# B&R Automation Studio project BatteryControl (part 3)

```iecst
	stepTest[0] := 50.000;
	stepTest[1] := 50.000;
	stepTest[2] := 50.000;
	stepTest[3] := 50.000;
	stepTest[4] := 50.000;
	stepTest[5] := 50.000;
	stepTest[6] := 50.000;
	stepTest[7] := 50.000;
	stepTest[8] := 50.000;
	stepTest[9] := 50.000;
	stepTest[10] := 50.010;
	stepTest[11] := 50.010;
	stepTest[12] := 50.010;
	stepTest[13] := 50.010;
	stepTest[14] := 50.010;
	stepTest[15] := 50.010;
	stepTest[16] := 50.010;
	stepTest[17] := 50.010;
	stepTest[18] := 50.010;
	stepTest[19] := 50.010;
	stepTest[20] := 50.010;
	stepTest[21] := 50.010;
	stepTest[22] := 50.010;
	stepTest[23] := 50.010;
	stepTest[24] := 50.010;
	stepTest[25] := 50.010;
	stepTest[26] := 50.010;
	stepTest[27] := 50.010;
	stepTest[28] := 50.010;
	stepTest[29] := 50.010;
	stepTest[30] := 50.010;
	stepTest[31] := 50.010;
	stepTest[32] := 50.010;
	stepTest[33] := 50.010;
	stepTest[34] := 50.010;
	stepTest[35] := 50.010;
	stepTest[36] := 50.010;
	stepTest[37] := 50.010;
	stepTest[38] := 50.010;
	stepTest[39] := 50.010;
	stepTest[40] := 50.000;
	stepTest[41] := 50.000;
	stepTest[42] := 50.000;
	stepTest[43] := 50.000;
	stepTest[44] := 50.000;
	stepTest[45] := 50.000;
	stepTest[46] := 50.000;
	stepTest[47] := 50.000;
	stepTest[48] := 50.000;
	stepTest[49] := 50.000;
	stepTest[50] := 49.990;
	stepTest[51] := 49.990;
	stepTest[52] := 49.990;
	stepTest[53] := 49.990;
	stepTest[54] := 49.990;
	stepTest[55] := 49.990;
	stepTest[56] := 49.990;
	stepTest[57] := 49.990;
	stepTest[58] := 49.990;
	stepTest[59] := 49.990;
	stepTest[60] := 49.990;
	stepTest[61] := 49.990;
	stepTest[62] := 49.990;
	stepTest[63] := 49.990;
	stepTest[64] := 49.990;
	stepTest[65] := 49.990;
	stepTest[66] := 49.990;
	stepTest[67] := 49.990;
	stepTest[68] := 49.990;
	stepTest[69] := 49.990;
	stepTest[70] := 49.990;
	stepTest[71] := 49.990;
	stepTest[72] := 49.990;
	stepTest[73] := 49.990;
	stepTest[74] := 49.990;
	stepTest[75] := 49.990;
	stepTest[76] := 49.990;
	stepTest[77] := 49.990;
	stepTest[78] := 49.990;
	stepTest[79] := 49.990;
	stepTest[80] := 50.000;
	stepTest[81] := 50.000;
	stepTest[82] := 50.000;
	stepTest[83] := 50.000;
	stepTest[84] := 50.000;
	stepTest[85] := 50.000;
	stepTest[86] := 50.000;
	stepTest[87] := 50.000;
	stepTest[88] := 50.000;
	stepTest[89] := 50.000;
	stepTest[90] := 50.020;
	stepTest[91] := 50.020;
	stepTest[92] := 50.020;
	stepTest[93] := 50.020;
	stepTest[94] := 50.020;
	stepTest[95] := 50.020;
	stepTest[96] := 50.020;
	stepTest[97] := 50.020;
	stepTest[98] := 50.020;
	stepTest[99] := 50.020;
	stepTest[100] := 50.020;
	stepTest[101] := 50.020;
	stepTest[102] := 50.020;
	stepTest[103] := 50.020;
	stepTest[104] := 50.020;
	stepTest[105] := 50.020;
	stepTest[106] := 50.020;
	stepTest[107] := 50.020;
	stepTest[108] := 50.020;
	stepTest[109] := 50.020;
	stepTest[110] := 50.020;
	stepTest[111] := 50.020;
	stepTest[112] := 50.020;
	stepTest[113] := 50.020;
	stepTest[114] := 50.020;
	stepTest[115] := 50.020;
	stepTest[116] := 50.020;
	stepTest[117] := 50.020;
	stepTest[118] := 50.020;
	stepTest[119] := 50.020;
	stepTest[120] := 50.000;
	stepTest[121] := 50.000;
	stepTest[122] := 50.000;
	stepTest[123] := 50.000;
	stepTest[124] := 50.000;
	stepTest[125] := 50.000;
	stepTest[126] := 50.000;
	stepTest[127] := 50.000;
	stepTest[128] := 50.000;
	stepTest[129] := 50.000;
	stepTest[130] := 49.980;
	stepTest[131] := 49.980;
	stepTest[132] := 49.980;
	stepTest[133] := 49.980;
	stepTest[134] := 49.980;
	stepTest[135] := 49.980;
	stepTest[136] := 49.980;
	stepTest[137] := 49.980;
	stepTest[138] := 49.980;
	stepTest[139] := 49.980;
	stepTest[140] := 49.980;
	stepTest[141] := 49.980;
	stepTest[142] := 49.980;
	stepTest[143] := 49.980;
	stepTest[144] := 49.980;
	stepTest[145] := 49.980;
	stepTest[146] := 49.980;
	stepTest[147] := 49.980;
	stepTest[148] := 49.980;
	stepTest[149] := 49.980;
	stepTest[150] := 49.980;
	stepTest[151] := 49.980;
	stepTest[152] := 49.980;
	stepTest[153] := 49.980;
	stepTest[154] := 49.980;
	stepTest[155] := 49.980;
	stepTest[156] := 49.980;
	stepTest[157] := 49.980;
	stepTest[158] := 49.980;
	stepTest[159] := 49.980;
	stepTest[160] := 50.000;
	stepTest[161] := 50.000;
	stepTest[162] := 50.000;
	stepTest[163] := 50.000;
	stepTest[164] := 50.000;
	stepTest[165] := 50.000;
	stepTest[166] := 50.000;
	stepTest[167] := 50.000;
	stepTest[168] := 50.000;
	stepTest[169] := 50.000;
	stepTest[170] := 50.100;
	stepTest[171] := 50.100;
	stepTest[172] := 50.100;
	stepTest[173] := 50.100;
	stepTest[174] := 50.100;
	stepTest[175] := 50.100;
	stepTest[176] := 50.100;
	stepTest[177] := 50.100;
	stepTest[178] := 50.100;
	stepTest[179] := 50.100;
	stepTest[180] := 50.100;
	stepTest[181] := 50.100;
	stepTest[182] := 50.100;
	stepTest[183] := 50.100;
	stepTest[184] := 50.100;
	stepTest[185] := 50.100;
	stepTest[186] := 50.100;
	stepTest[187] := 50.100;
	stepTest[188] := 50.100;
	stepTest[189] := 50.100;
	stepTest[190] := 50.100;
	stepTest[191] := 50.100;
	stepTest[192] := 50.100;
	stepTest[193] := 50.100;
	stepTest[194] := 50.100;
	stepTest[195] := 50.100;
	stepTest[196] := 50.100;
	stepTest[197] := 50.100;
	stepTest[198] := 50.100;
	stepTest[199] := 50.100;
	stepTest[200] := 50.000;
	stepTest[201] := 50.000;
	stepTest[202] := 50.000;
	stepTest[203] := 50.000;
	stepTest[204] := 50.000;
	stepTest[205] := 50.000;
	stepTest[206] := 50.000;
	stepTest[207] := 50.000;
	stepTest[208] := 50.000;
	stepTest[209] := 50.000;
	stepTest[210] := 49.900;
	stepTest[211] := 49.900;
	stepTest[212] := 49.900;
	stepTest[213] := 49.900;
	stepTest[214] := 49.900;
	stepTest[215] := 49.900;
	stepTest[216] := 49.900;
	stepTest[217] := 49.900;
	stepTest[218] := 49.900;
	stepTest[219] := 49.900;
	stepTest[220] := 49.900;
	stepTest[221] := 49.900;
	stepTest[222] := 49.900;
	stepTest[223] := 49.900;
	stepTest[224] := 49.900;
	stepTest[225] := 49.900;
	stepTest[226] := 49.900;
	stepTest[227] := 49.900;
	stepTest[228] := 49.900;
	stepTest[229] := 49.900;
	stepTest[230] := 49.900;
	stepTest[231] := 49.900;
	stepTest[232] := 49.900;
	stepTest[233] := 49.900;
	stepTest[234] := 49.900;
	stepTest[235] := 49.900;
	stepTest[236] := 49.900;
	stepTest[237] := 49.900;
	stepTest[238] := 49.900;
	stepTest[239] := 49.900;
	stepTest[240] := 50.000;
	stepTest[241] := 50.000;
	stepTest[242] := 50.000;
	stepTest[243] := 50.000;
	stepTest[244] := 50.000;
	stepTest[245] := 50.000;
	stepTest[246] := 50.000;
	stepTest[247] := 50.000;
	stepTest[248] := 50.000;
	stepTest[249] := 50.000;
	stepTest[250] := 50.200;
	stepTest[251] := 50.200;
	stepTest[252] := 50.200;
	stepTest[253] := 50.200;
	stepTest[254] := 50.200;
	stepTest[255] := 50.200;
	stepTest[256] := 50.200;
	stepTest[257] := 50.200;
	stepTest[258] := 50.200;
	stepTest[259] := 50.200;
	stepTest[260] := 50.200;
	stepTest[261] := 50.200;
	stepTest[262] := 50.200;
	stepTest[263] := 50.200;
	stepTest[264] := 50.200;
	stepTest[265] := 50.200;
	stepTest[266] := 50.200;
	stepTest[267] := 50.200;
	stepTest[268] := 50.200;
	stepTest[269] := 50.200;
	stepTest[270] := 50.200;
	stepTest[271] := 50.200;
	stepTest[272] := 50.200;
	stepTest[273] := 50.200;
	stepTest[274] := 50.200;
	stepTest[275] := 50.200;
	stepTest[276] := 50.200;
	stepTest[277] := 50.200;
	stepTest[278] := 50.200;
	stepTest[279] := 50.200;
	stepTest[280] := 50.000;
	stepTest[281] := 50.000;
	stepTest[282] := 50.000;
	stepTest[283] := 50.000;
	stepTest[284] := 50.000;
	stepTest[285] := 50.000;
	stepTest[286] := 50.000;
	stepTest[287] := 50.000;
	stepTest[288] := 50.000;
	stepTest[289] := 50.000;
	stepTest[290] := 49.800;
	stepTest[291] := 49.800;
	stepTest[292] := 49.800;
	stepTest[293] := 49.800;
	stepTest[294] := 49.800;
	stepTest[295] := 49.800;
	stepTest[296] := 49.800;
	stepTest[297] := 49.800;
	stepTest[298] := 49.800;
	stepTest[299] := 49.800;
	stepTest[300] := 49.800;
	stepTest[301] := 49.800;
	stepTest[302] := 49.800;
	stepTest[303] := 49.800;
	stepTest[304] := 49.800;
	stepTest[305] := 49.800;
	stepTest[306] := 49.800;
	stepTest[307] := 49.800;
	stepTest[308] := 49.800;
	stepTest[309] := 49.800;
	stepTest[310] := 49.800;
	stepTest[311] := 49.800;
	stepTest[312] := 49.800;
	stepTest[313] := 49.800;
	stepTest[314] := 49.800;
	stepTest[315] := 49.800;
	stepTest[316] := 49.800;
	stepTest[317] := 49.800;
	stepTest[318] := 49.800;
	stepTest[319] := 49.800;
	stepTest[320] := 50.000;
	stepTest[321] := 50.000;
	stepTest[322] := 50.000;
	stepTest[323] := 50.000;
	stepTest[324] := 50.000;
	stepTest[325] := 50.000;
	stepTest[326] := 50.000;
	stepTest[327] := 50.000;
	stepTest[328] := 50.000;
	stepTest[329] := 50.000;
	stepTest[330] := 50.300;
	stepTest[331] := 50.300;
	stepTest[332] := 50.300;
	stepTest[333] := 50.300;
	stepTest[334] := 50.300;
	stepTest[335] := 50.300;
	stepTest[336] := 50.300;
	stepTest[337] := 50.300;
	stepTest[338] := 50.300;
	stepTest[339] := 50.300;
	stepTest[340] := 50.300;
	stepTest[341] := 50.300;
	stepTest[342] := 50.300;
	stepTest[343] := 50.300;
	stepTest[344] := 50.300;
	stepTest[345] := 50.300;
	stepTest[346] := 50.300;
	stepTest[347] := 50.300;
	stepTest[348] := 50.300;
	stepTest[349] := 50.300;
	stepTest[350] := 50.300;
	stepTest[351] := 50.300;
	stepTest[352] := 50.300;
	stepTest[353] := 50.300;
	stepTest[354] := 50.300;
	stepTest[355] := 50.300;
	stepTest[356] := 50.300;
	stepTest[357] := 50.300;
	stepTest[358] := 50.300;
	stepTest[359] := 50.300;
	stepTest[360] := 50.000;
	stepTest[361] := 50.000;
	stepTest[362] := 50.000;
	stepTest[363] := 50.000;
	stepTest[364] := 50.000;
	stepTest[365] := 50.000;
	stepTest[366] := 50.000;
	stepTest[367] := 50.000;
	stepTest[368] := 50.000;
	stepTest[369] := 50.000;
	stepTest[370] := 49.700;
	stepTest[371] := 49.700;
	stepTest[372] := 49.700;
	stepTest[373] := 49.700;
	stepTest[374] := 49.700;
	stepTest[375] := 49.700;
	stepTest[376] := 49.700;
	stepTest[377] := 49.700;
	stepTest[378] := 49.700;
	stepTest[379] := 49.700;
	stepTest[380] := 49.700;
	stepTest[381] := 49.700;
	stepTest[382] := 49.700;
	stepTest[383] := 49.700;
	stepTest[384] := 49.700;
	stepTest[385] := 49.700;
	stepTest[386] := 49.700;
	stepTest[387] := 49.700;
	stepTest[388] := 49.700;
	stepTest[389] := 49.700;
	stepTest[390] := 49.700;
	stepTest[391] := 49.700;
	stepTest[392] := 49.700;
	stepTest[393] := 49.700;
	stepTest[394] := 49.700;
	stepTest[395] := 49.700;
	stepTest[396] := 49.700;
	stepTest[397] := 49.700;
	stepTest[398] := 49.700;
	stepTest[399] := 49.700;
	stepTest[400] := 50.000;
	stepTest[401] := 50.000;
	stepTest[402] := 50.000;
	stepTest[403] := 50.000;
	stepTest[404] := 50.000;
	stepTest[405] := 50.000;
	stepTest[406] := 50.000;
	stepTest[407] := 50.000;
	stepTest[408] := 50.000;
	stepTest[409] := 50.000;
	stepTest[410] := 50.400;
	stepTest[411] := 50.400;
	stepTest[412] := 50.400;
	stepTest[413] := 50.400;
	stepTest[414] := 50.400;
	stepTest[415] := 50.400;
	stepTest[416] := 50.400;
	stepTest[417] := 50.400;
	stepTest[418] := 50.400;
	stepTest[419] := 50.400;
	stepTest[420] := 50.400;
	stepTest[421] := 50.400;
	stepTest[422] := 50.400;
	stepTest[423] := 50.400;
	stepTest[424] := 50.400;
	stepTest[425] := 50.400;
	stepTest[426] := 50.400;
	stepTest[427] := 50.400;
	stepTest[428] := 50.400;
	stepTest[429] := 50.400;
	stepTest[430] := 50.400;
	stepTest[431] := 50.400;
	stepTest[432] := 50.400;
	stepTest[433] := 50.400;
	stepTest[434] := 50.400;
	stepTest[435] := 50.400;
	stepTest[436] := 50.400;
	stepTest[437] := 50.400;
	stepTest[438] := 50.400;
	stepTest[439] := 50.400;
	stepTest[440] := 50.000;
	stepTest[441] := 50.000;
	stepTest[442] := 50.000;
	stepTest[443] := 50.000;
	stepTest[444] := 50.000;
	stepTest[445] := 50.000;
	stepTest[446] := 50.000;
	stepTest[447] := 50.000;
	stepTest[448] := 50.000;
	stepTest[449] := 50.000;
	stepTest[450] := 49.600;
	stepTest[451] := 49.600;
	stepTest[452] := 49.600;
	stepTest[453] := 49.600;
	stepTest[454] := 49.600;
	stepTest[455] := 49.600;
	stepTest[456] := 49.600;
	stepTest[457] := 49.600;
	stepTest[458] := 49.600;
	stepTest[459] := 49.600;
	stepTest[460] := 49.600;
	stepTest[461] := 49.600;
	stepTest[462] := 49.600;
	stepTest[463] := 49.600;
	stepTest[464] := 49.600;
	stepTest[465] := 49.600;
	stepTest[466] := 49.600;
	stepTest[467] := 49.600;
	stepTest[468] := 49.600;
	stepTest[469] := 49.600;
	stepTest[470] := 49.600;
	stepTest[471] := 49.600;
	stepTest[472] := 49.600;
	stepTest[473] := 49.600;
	stepTest[474] := 49.600;
	stepTest[475] := 49.600;
	stepTest[476] := 49.600;
	stepTest[477] := 49.600;
	stepTest[478] := 49.600;
	stepTest[479] := 49.600;
	stepTest[480] := 50.000;
	stepTest[481] := 50.000;
	stepTest[482] := 50.000;
	stepTest[483] := 50.000;
	stepTest[484] := 50.000;
	stepTest[485] := 50.000;
	stepTest[486] := 50.000;
	stepTest[487] := 50.000;
	stepTest[488] := 50.000;
	stepTest[489] := 50.000;
	stepTest[490] := 50.500;
	stepTest[491] := 50.500;
	stepTest[492] := 50.500;
	stepTest[493] := 50.500;
	stepTest[494] := 50.500;
	stepTest[495] := 50.500;
	stepTest[496] := 50.500;
	stepTest[497] := 50.500;
	stepTest[498] := 50.500;
	stepTest[499] := 50.500;
	stepTest[500] := 50.500;
	stepTest[501] := 50.500;
	stepTest[502] := 50.500;
	stepTest[503] := 50.500;
	stepTest[504] := 50.500;
	stepTest[505] := 50.500;
	stepTest[506] := 50.500;
	stepTest[507] := 50.500;
	stepTest[508] := 50.500;
	stepTest[509] := 50.500;
	stepTest[510] := 50.500;
	stepTest[511] := 50.500;
	stepTest[512] := 50.500;
	stepTest[513] := 50.500;
	stepTest[514] := 50.500;
	stepTest[515] := 50.500;
	stepTest[516] := 50.500;
	stepTest[517] := 50.500;
	stepTest[518] := 50.500;
	stepTest[519] := 50.500;
	stepTest[520] := 50.000;
	stepTest[521] := 50.000;
	stepTest[522] := 50.000;
	stepTest[523] := 50.000;
	stepTest[524] := 50.000;
	stepTest[525] := 50.000;
	stepTest[526] := 50.000;
	stepTest[527] := 50.000;
	stepTest[528] := 50.000;
	stepTest[529] := 50.000;
	stepTest[530] := 49.500;
	stepTest[531] := 49.500;
	stepTest[532] := 49.500;
	stepTest[533] := 49.500;
	stepTest[534] := 49.500;
	stepTest[535] := 49.500;
	stepTest[536] := 49.500;
	stepTest[537] := 49.500;
	stepTest[538] := 49.500;
	stepTest[539] := 49.500;
	stepTest[540] := 49.500;
	stepTest[541] := 49.500;
	stepTest[542] := 49.500;
	stepTest[543] := 49.500;
	stepTest[544] := 49.500;
	stepTest[545] := 49.500;
	stepTest[546] := 49.500;
	stepTest[547] := 49.500;
	stepTest[548] := 49.500;
	stepTest[549] := 49.500;
	stepTest[550] := 49.500;
	stepTest[551] := 49.500;
	stepTest[552] := 49.500;
	stepTest[553] := 49.500;
	stepTest[554] := 49.500;
	stepTest[555] := 49.500;
	stepTest[556] := 49.500;
	stepTest[557] := 49.500;
	stepTest[558] := 49.500;
	stepTest[559] := 49.500;
	stepTest[560] := 50.000;
	stepTest[561] := 50.000;
	stepTest[562] := 50.000;
	stepTest[563] := 50.000;
	stepTest[564] := 50.000;
	stepTest[565] := 50.000;
	stepTest[566] := 50.000;
	stepTest[567] := 50.000;
	stepTest[568] := 50.000;
	stepTest[569] := 50.000;

	sustainLF[0]:=50.000;
	sustainLF[1]:=50.000;
	sustainLF[2]:=50.000;
	sustainLF[3]:=50.000;
	sustainLF[4]:=50.000;
	sustainLF[5]:=50.000;
	sustainLF[6]:=50.000;
	sustainLF[7]:=50.000;
	sustainLF[8]:=50.000;
	sustainLF[9]:=50.000;
	sustainLF[10]:=50.000;
	sustainLF[11]:=50.000;
	sustainLF[12]:=50.000;
	sustainLF[13]:=50.000;
	sustainLF[14]:=50.000;
	sustainLF[15]:=50.000;
	sustainLF[16]:=50.000;
	sustainLF[17]:=50.000;
	sustainLF[18]:=50.000;
	sustainLF[19]:=50.000;
	sustainLF[20]:=50.000;
	sustainLF[21]:=50.000;
	sustainLF[22]:=50.000;
	sustainLF[23]:=50.000;
	sustainLF[24]:=50.000;
	sustainLF[25]:=50.000;
	sustainLF[26]:=50.000;
	sustainLF[27]:=50.000;
	sustainLF[28]:=50.000;
	sustainLF[29]:=50.000;
	sustainLF[30]:=49.400;
	sustainLF[31]:=49.400;
	sustainLF[32]:=49.400;
	sustainLF[33]:=49.400;
	sustainLF[34]:=49.400;
	sustainLF[35]:=49.400;
	sustainLF[36]:=49.400;
	sustainLF[37]:=49.400;
	sustainLF[38]:=49.400;
	sustainLF[39]:=49.400;
	sustainLF[40]:=49.400;
	sustainLF[41]:=49.400;
	sustainLF[42]:=49.400;
	sustainLF[43]:=49.400;
	sustainLF[44]:=49.400;
	sustainLF[45]:=49.400;
	sustainLF[46]:=49.400;
	sustainLF[47]:=49.400;
	sustainLF[48]:=49.400;
	sustainLF[49]:=49.400;
	sustainLF[50]:=49.400;
	sustainLF[51]:=49.400;
	sustainLF[52]:=49.400;
	sustainLF[53]:=49.400;
	sustainLF[54]:=49.400;
	sustainLF[55]:=49.400;
	sustainLF[56]:=49.400;
	sustainLF[57]:=49.400;
	sustainLF[58]:=49.400;
	sustainLF[59]:=49.400;
	sustainLF[60]:=49.400;
	sustainLF[61]:=49.400;
	sustainLF[62]:=49.400;
	sustainLF[63]:=49.400;
	sustainLF[64]:=49.400;
	sustainLF[65]:=49.400;
	sustainLF[66]:=49.400;
	sustainLF[67]:=49.400;
	sustainLF[68]:=49.400;
	sustainLF[69]:=49.400;
	sustainLF[70]:=49.400;
	sustainLF[71]:=49.400;
	sustainLF[72]:=49.400;
	sustainLF[73]:=49.400;
	sustainLF[74]:=49.400;
	sustainLF[75]:=49.400;
	sustainLF[76]:=49.400;
	sustainLF[77]:=49.400;
	sustainLF[78]:=49.400;
	sustainLF[79]:=49.400;
	sustainLF[80]:=49.400;
	sustainLF[81]:=49.400;
	sustainLF[82]:=49.400;
	sustainLF[83]:=49.400;
	sustainLF[84]:=49.400;
	sustainLF[85]:=49.400;
	sustainLF[86]:=49.400;
	sustainLF[87]:=49.400;
	sustainLF[88]:=49.400;
	sustainLF[89]:=49.400;
	sustainLF[90]:=49.400;
	sustainLF[91]:=49.400;
	sustainLF[92]:=49.400;
	sustainLF[93]:=49.400;
	sustainLF[94]:=49.400;
	sustainLF[95]:=49.400;
	sustainLF[96]:=49.400;
	sustainLF[97]:=49.400;
	sustainLF[98]:=49.400;
	sustainLF[99]:=49.400;
	sustainLF[100]:=49.400;
	sustainLF[101]:=49.400;
	sustainLF[102]:=49.400;
	sustainLF[103]:=49.400;
	sustainLF[104]:=49.400;
	sustainLF[105]:=49.400;
	sustainLF[106]:=49.400;
	sustainLF[107]:=49.400;
	sustainLF[108]:=49.400;
	sustainLF[109]:=49.400;
	sustainLF[110]:=49.400;
	sustainLF[111]:=49.400;
	sustainLF[112]:=49.400;
	sustainLF[113]:=49.400;
	sustainLF[114]:=49.400;
	sustainLF[115]:=49.400;
	sustainLF[116]:=49.400;
	sustainLF[117]:=49.400;
	sustainLF[118]:=49.400;
	sustainLF[119]:=49.400;
	sustainLF[120]:=49.400;
	sustainLF[121]:=49.400;
	sustainLF[122]:=49.400;
	sustainLF[123]:=49.400;
	sustainLF[124]:=49.400;
	sustainLF[125]:=49.400;
	sustainLF[126]:=49.400;
	sustainLF[127]:=49.400;
	sustainLF[128]:=49.400;
	sustainLF[129]:=49.400;
	sustainLF[130]:=49.400;
	sustainLF[131]:=49.400;
	sustainLF[132]:=49.400;
	sustainLF[133]:=49.400;
	sustainLF[134]:=49.400;
	sustainLF[135]:=49.400;
	sustainLF[136]:=49.400;
	sustainLF[137]:=49.400;
	sustainLF[138]:=49.400;
	sustainLF[139]:=49.400;
	sustainLF[140]:=49.400;
	sustainLF[141]:=49.400;
	sustainLF[142]:=49.400;
	sustainLF[143]:=49.400;
	sustainLF[144]:=49.400;
	sustainLF[145]:=49.400;
	sustainLF[146]:=49.400;
	sustainLF[147]:=49.400;
	sustainLF[148]:=49.400;
	sustainLF[149]:=49.400;
	sustainLF[150]:=49.400;
	sustainLF[151]:=49.400;
	sustainLF[152]:=49.400;
	sustainLF[153]:=49.400;
	sustainLF[154]:=49.400;
	sustainLF[155]:=49.400;
	sustainLF[156]:=49.400;
	sustainLF[157]:=49.400;
	sustainLF[158]:=49.400;
	sustainLF[159]:=49.400;
	sustainLF[160]:=49.400;
	sustainLF[161]:=49.400;
	sustainLF[162]:=49.400;
	sustainLF[163]:=49.400;
	sustainLF[164]:=49.400;
	sustainLF[165]:=49.400;
	sustainLF[166]:=49.400;
	sustainLF[167]:=49.400;
	sustainLF[168]:=49.400;
	sustainLF[169]:=49.400;
	sustainLF[170]:=49.400;
	sustainLF[171]:=49.400;
	sustainLF[172]:=49.400;
	sustainLF[173]:=49.400;
	sustainLF[174]:=49.400;
	sustainLF[175]:=49.400;
	sustainLF[176]:=49.400;
	sustainLF[177]:=49.400;
	sustainLF[178]:=49.400;
	sustainLF[179]:=49.400;
	sustainLF[180]:=49.400;
	sustainLF[181]:=49.400;
	sustainLF[182]:=49.400;
	sustainLF[183]:=49.400;
	sustainLF[184]:=49.400;
	sustainLF[185]:=49.400;
	sustainLF[186]:=49.400;
	sustainLF[187]:=49.400;
	sustainLF[188]:=49.400;
	sustainLF[189]:=49.400;
	sustainLF[190]:=49.400;
	sustainLF[191]:=49.400;
	sustainLF[192]:=49.400;
	sustainLF[193]:=49.400;
	sustainLF[194]:=49.400;
	sustainLF[195]:=49.400;
	sustainLF[196]:=49.400;
	sustainLF[197]:=49.400;
	sustainLF[198]:=49.400;
	sustainLF[199]:=49.400;
	sustainLF[200]:=49.400;
	sustainLF[201]:=49.400;
	sustainLF[202]:=49.400;
	sustainLF[203]:=49.400;
	sustainLF[204]:=49.400;
	sustainLF[205]:=49.400;
	sustainLF[206]:=49.400;
	sustainLF[207]:=49.400;
	sustainLF[208]:=49.400;
	sustainLF[209]:=49.400;
	sustainLF[210]:=49.400;
	sustainLF[211]:=49.400;
	sustainLF[212]:=49.400;
	sustainLF[213]:=49.400;
	sustainLF[214]:=49.400;
	sustainLF[215]:=49.400;
	sustainLF[216]:=49.400;
	sustainLF[217]:=49.400;
	sustainLF[218]:=49.400;
	sustainLF[219]:=49.400;
	sustainLF[220]:=49.400;
	sustainLF[221]:=49.400;
	sustainLF[222]:=49.400;
	sustainLF[223]:=49.400;
	sustainLF[224]:=49.400;
	sustainLF[225]:=49.400;
	sustainLF[226]:=49.400;
	sustainLF[227]:=49.400;
	sustainLF[228]:=49.400;
	sustainLF[229]:=49.400;
	sustainLF[230]:=49.400;
	sustainLF[231]:=49.400;
	sustainLF[232]:=49.400;
	sustainLF[233]:=49.400;
	sustainLF[234]:=49.400;
	sustainLF[235]:=49.400;
	sustainLF[236]:=49.400;
	sustainLF[237]:=49.400;
	sustainLF[238]:=49.400;
	sustainLF[239]:=49.400;
	sustainLF[240]:=49.400;
	sustainLF[241]:=49.400;
	sustainLF[242]:=49.400;
	sustainLF[243]:=49.400;
	sustainLF[244]:=49.400;
	sustainLF[245]:=49.400;
	sustainLF[246]:=49.400;
	sustainLF[247]:=49.400;
	sustainLF[248]:=49.400;
	sustainLF[249]:=49.400;
	sustainLF[250]:=49.400;
	sustainLF[251]:=49.400;
	sustainLF[252]:=49.400;
	sustainLF[253]:=49.400;
	sustainLF[254]:=49.400;
	sustainLF[255]:=49.400;
	sustainLF[256]:=49.400;
	sustainLF[257]:=49.400;
	sustainLF[258]:=49.400;
	sustainLF[259]:=49.400;
	sustainLF[260]:=49.400;
	sustainLF[261]:=49.400;
	sustainLF[262]:=49.400;
	sustainLF[263]:=49.400;
	sustainLF[264]:=49.400;
	sustainLF[265]:=49.400;
	sustainLF[266]:=49.400;
	sustainLF[267]:=49.400;
	sustainLF[268]:=49.400;
	sustainLF[269]:=49.400;
	sustainLF[270]:=49.400;
	sustainLF[271]:=49.400;
	sustainLF[272]:=49.400;
	sustainLF[273]:=49.400;
	sustainLF[274]:=49.400;
	sustainLF[275]:=49.400;
	sustainLF[276]:=49.400;
	sustainLF[277]:=49.400;
	sustainLF[278]:=49.400;
	sustainLF[279]:=49.400;
	sustainLF[280]:=49.400;
	sustainLF[281]:=49.400;
	sustainLF[282]:=49.400;
	sustainLF[283]:=49.400;
	sustainLF[284]:=49.400;
	sustainLF[285]:=49.400;
	sustainLF[286]:=49.400;
	sustainLF[287]:=49.400;
	sustainLF[288]:=49.400;
	sustainLF[289]:=49.400;
	sustainLF[290]:=49.400;
	sustainLF[291]:=49.400;
	sustainLF[292]:=49.400;
	sustainLF[293]:=49.400;
	sustainLF[294]:=49.400;
	sustainLF[295]:=49.400;
	sustainLF[296]:=49.400;
	sustainLF[297]:=49.400;
	sustainLF[298]:=49.400;
	sustainLF[299]:=49.400;
	sustainLF[300]:=49.400;
	sustainLF[301]:=49.400;
	sustainLF[302]:=49.400;
	sustainLF[303]:=49.400;
	sustainLF[304]:=49.400;
	sustainLF[305]:=49.400;
	sustainLF[306]:=49.400;
	sustainLF[307]:=49.400;
	sustainLF[308]:=49.400;
	sustainLF[309]:=49.400;
	sustainLF[310]:=49.400;
	sustainLF[311]:=49.400;
	sustainLF[312]:=49.400;
	sustainLF[313]:=49.400;
	sustainLF[314]:=49.400;
	sustainLF[315]:=49.400;
	sustainLF[316]:=49.400;
	sustainLF[317]:=49.400;
	sustainLF[318]:=49.400;
	sustainLF[319]:=49.400;
	sustainLF[320]:=49.400;
	sustainLF[321]:=49.400;
	sustainLF[322]:=49.400;
	sustainLF[323]:=49.400;
	sustainLF[324]:=49.400;
	sustainLF[325]:=49.400;
	sustainLF[326]:=49.400;
	sustainLF[327]:=49.400;
	sustainLF[328]:=49.400;
	sustainLF[329]:=49.400;
	sustainLF[330]:=49.400;
	sustainLF[331]:=49.400;
	sustainLF[332]:=49.400;
	sustainLF[333]:=49.400;
	sustainLF[334]:=49.400;
	sustainLF[335]:=49.400;
	sustainLF[336]:=49.400;
	sustainLF[337]:=49.400;
	sustainLF[338]:=49.400;
	sustainLF[339]:=49.400;
	sustainLF[340]:=49.400;
	sustainLF[341]:=49.400;
	sustainLF[342]:=49.400;
	sustainLF[343]:=49.400;
	sustainLF[344]:=49.400;
	sustainLF[345]:=49.400;
	sustainLF[346]:=49.400;
	sustainLF[347]:=49.400;
	sustainLF[348]:=49.400;
	sustainLF[349]:=49.400;
	sustainLF[350]:=49.400;
	sustainLF[351]:=49.400;
	sustainLF[352]:=49.400;
	sustainLF[353]:=49.400;
	sustainLF[354]:=49.400;
	sustainLF[355]:=49.400;
	sustainLF[356]:=49.400;
	sustainLF[357]:=49.400;
	sustainLF[358]:=49.400;
	sustainLF[359]:=49.400;
	sustainLF[360]:=49.400;
	sustainLF[361]:=49.400;
	sustainLF[362]:=49.400;
	sustainLF[363]:=49.400;
	sustainLF[364]:=49.400;
	sustainLF[365]:=49.400;
	sustainLF[366]:=49.400;
	sustainLF[367]:=49.400;
	sustainLF[368]:=49.400;
	sustainLF[369]:=49.400;
	sustainLF[370]:=49.400;
	sustainLF[371]:=49.400;
	sustainLF[372]:=49.400;
	sustainLF[373]:=49.400;
	sustainLF[374]:=49.400;
	sustainLF[375]:=49.400;
	sustainLF[376]:=49.400;
	sustainLF[377]:=49.400;
	sustainLF[378]:=49.400;
	sustainLF[379]:=49.400;
	sustainLF[380]:=49.400;
	sustainLF[381]:=49.400;
	sustainLF[382]:=49.400;
	sustainLF[383]:=49.400;
	sustainLF[384]:=49.400;
	sustainLF[385]:=49.400;
	sustainLF[386]:=49.400;
	sustainLF[387]:=49.400;
	sustainLF[388]:=49.400;
	sustainLF[389]:=49.400;
	sustainLF[390]:=49.400;
	sustainLF[391]:=49.400;
	sustainLF[392]:=49.400;
	sustainLF[393]:=49.400;
	sustainLF[394]:=49.400;
	sustainLF[395]:=49.400;
	sustainLF[396]:=49.400;
	sustainLF[397]:=49.400;
	sustainLF[398]:=49.400;
	sustainLF[399]:=49.400;
	sustainLF[400]:=49.400;
	sustainLF[401]:=49.400;
	sustainLF[402]:=49.400;
	sustainLF[403]:=49.400;
	sustainLF[404]:=49.400;
	sustainLF[405]:=49.400;
	sustainLF[406]:=49.400;
	sustainLF[407]:=49.400;
	sustainLF[408]:=49.400;
	sustainLF[409]:=49.400;
	sustainLF[410]:=49.400;
	sustainLF[411]:=49.400;
	sustainLF[412]:=49.400;
	sustainLF[413]:=49.400;
	sustainLF[414]:=49.400;
	sustainLF[415]:=49.400;
	sustainLF[416]:=49.400;
	sustainLF[417]:=49.400;
	sustainLF[418]:=49.400;
	sustainLF[419]:=49.400;
	sustainLF[420]:=49.400;
	sustainLF[421]:=49.400;
	sustainLF[422]:=49.400;
	sustainLF[423]:=49.400;
	sustainLF[424]:=49.400;
	sustainLF[425]:=49.400;
	sustainLF[426]:=49.400;
	sustainLF[427]:=49.400;
	sustainLF[428]:=49.400;
	sustainLF[429]:=49.400;
	sustainLF[430]:=49.400;
	sustainLF[431]:=49.400;
	sustainLF[432]:=49.400;
	sustainLF[433]:=49.400;
	sustainLF[434]:=49.400;
	sustainLF[435]:=49.400;
	sustainLF[436]:=49.400;
	sustainLF[437]:=49.400;
	sustainLF[438]:=49.400;
	sustainLF[439]:=49.400;
	sustainLF[440]:=49.400;
	sustainLF[441]:=49.400;
	sustainLF[442]:=49.400;
	sustainLF[443]:=49.400;
	sustainLF[444]:=49.400;
	sustainLF[445]:=49.400;
	sustainLF[446]:=49.400;
	sustainLF[447]:=49.400;
	sustainLF[448]:=49.400;
	sustainLF[449]:=49.400;
	sustainLF[450]:=49.400;
	sustainLF[451]:=49.400;
	sustainLF[452]:=49.400;
	sustainLF[453]:=49.400;
	sustainLF[454]:=49.400;
	sustainLF[455]:=49.400;
	sustainLF[456]:=49.400;
	sustainLF[457]:=49.400;
	sustainLF[458]:=49.400;
	sustainLF[459]:=49.400;
	sustainLF[460]:=49.400;
	sustainLF[461]:=49.400;
	sustainLF[462]:=49.400;
	sustainLF[463]:=49.400;
	sustainLF[464]:=49.400;
	sustainLF[465]:=49.400;
	sustainLF[466]:=49.400;
	sustainLF[467]:=49.400;
	sustainLF[468]:=49.400;
	sustainLF[469]:=49.400;
	sustainLF[470]:=49.400;
	sustainLF[471]:=49.400;
	sustainLF[472]:=49.400;
	sustainLF[473]:=49.400;
	sustainLF[474]:=49.400;
	sustainLF[475]:=49.400;
	sustainLF[476]:=49.400;
	sustainLF[477]:=49.400;
	sustainLF[478]:=49.400;
	sustainLF[479]:=49.400;
	sustainLF[480]:=49.400;
	sustainLF[481]:=49.400;
	sustainLF[482]:=49.400;
	sustainLF[483]:=49.400;
	sustainLF[484]:=49.400;
	sustainLF[485]:=49.400;
	sustainLF[486]:=49.400;
	sustainLF[487]:=49.400;
	sustainLF[488]:=49.400;
	sustainLF[489]:=49.400;
	sustainLF[490]:=49.400;
	sustainLF[491]:=49.400;
	sustainLF[492]:=49.400;
	sustainLF[493]:=49.400;
	sustainLF[494]:=49.400;
	sustainLF[495]:=49.400;
	sustainLF[496]:=49.400;
	sustainLF[497]:=49.400;
	sustainLF[498]:=49.400;
	sustainLF[499]:=49.400;
	sustainLF[500]:=49.400;
	sustainLF[501]:=49.400;
	sustainLF[502]:=49.400;
	sustainLF[503]:=49.400;
	sustainLF[504]:=49.400;
	sustainLF[505]:=49.400;
	sustainLF[506]:=49.400;
	sustainLF[507]:=49.400;
	sustainLF[508]:=49.400;
	sustainLF[509]:=49.400;
	sustainLF[510]:=49.400;
	sustainLF[511]:=49.400;
	sustainLF[512]:=49.400;
	sustainLF[513]:=49.400;
	sustainLF[514]:=49.400;
	sustainLF[515]:=49.400;
	sustainLF[516]:=49.400;
	sustainLF[517]:=49.400;
	sustainLF[518]:=49.400;
	sustainLF[519]:=49.400;
	sustainLF[520]:=49.400;
	sustainLF[521]:=49.400;
	sustainLF[522]:=49.400;
	sustainLF[523]:=49.400;
	sustainLF[524]:=49.400;
	sustainLF[525]:=49.400;
	sustainLF[526]:=49.400;
	sustainLF[527]:=49.400;
	sustainLF[528]:=49.400;
	sustainLF[529]:=49.400;
	sustainLF[530]:=49.400;
	sustainLF[531]:=49.400;
	sustainLF[532]:=49.400;
	sustainLF[533]:=49.400;
	sustainLF[534]:=49.400;
	sustainLF[535]:=49.400;
	sustainLF[536]:=49.400;
	sustainLF[537]:=49.400;
	sustainLF[538]:=49.400;
	sustainLF[539]:=49.400;
	sustainLF[540]:=49.400;
	sustainLF[541]:=49.400;
	sustainLF[542]:=49.400;
	sustainLF[543]:=49.400;
	sustainLF[544]:=49.400;
	sustainLF[545]:=49.400;
	sustainLF[546]:=49.400;
	sustainLF[547]:=49.400;
	sustainLF[548]:=49.400;
	sustainLF[549]:=49.400;
	sustainLF[550]:=49.400;
	sustainLF[551]:=49.400;
	sustainLF[552]:=49.400;
	sustainLF[553]:=49.400;
	sustainLF[554]:=49.400;
	sustainLF[555]:=49.400;
	sustainLF[556]:=49.400;
	sustainLF[557]:=49.400;
	sustainLF[558]:=49.400;
	sustainLF[559]:=49.400;
	sustainLF[560]:=49.400;
	sustainLF[561]:=49.400;
	sustainLF[562]:=49.400;
	sustainLF[563]:=49.400;
	sustainLF[564]:=49.400;
	sustainLF[565]:=49.400;
	sustainLF[566]:=49.400;
	sustainLF[567]:=49.400;
	sustainLF[568]:=49.400;
	sustainLF[569]:=49.400;
	sustainLF[570]:=49.400;
	sustainLF[571]:=49.400;
	sustainLF[572]:=49.400;
	sustainLF[573]:=49.400;
	sustainLF[574]:=49.400;
	sustainLF[575]:=49.400;
	sustainLF[576]:=49.400;
	sustainLF[577]:=49.400;
	sustainLF[578]:=49.400;
	sustainLF[579]:=49.400;
	sustainLF[580]:=49.400;
	sustainLF[581]:=49.400;
	sustainLF[582]:=49.400;
	sustainLF[583]:=49.400;
	sustainLF[584]:=49.400;
	sustainLF[585]:=49.400;
	sustainLF[586]:=49.400;
	sustainLF[587]:=49.400;
	sustainLF[588]:=49.400;
	sustainLF[589]:=49.400;
	sustainLF[590]:=49.400;
	sustainLF[591]:=49.400;
	sustainLF[592]:=49.400;
	sustainLF[593]:=49.400;
	sustainLF[594]:=49.400;
	sustainLF[595]:=49.400;
	sustainLF[596]:=49.400;
	sustainLF[597]:=49.400;
	sustainLF[598]:=49.400;
	sustainLF[599]:=49.400;
	sustainLF[600]:=49.400;
	sustainLF[601]:=49.400;
	sustainLF[602]:=49.400;
	sustainLF[603]:=49.400;
	sustainLF[604]:=49.400;
	sustainLF[605]:=49.400;
	sustainLF[606]:=49.400;
	sustainLF[607]:=49.400;
	sustainLF[608]:=49.400;
	sustainLF[609]:=49.400;
	sustainLF[610]:=49.400;
	sustainLF[611]:=49.400;
	sustainLF[612]:=49.400;
	sustainLF[613]:=49.400;
	sustainLF[614]:=49.400;
	sustainLF[615]:=49.400;
	sustainLF[616]:=49.400;
	sustainLF[617]:=49.400;
	sustainLF[618]:=49.400;
	sustainLF[619]:=49.400;
	sustainLF[620]:=49.400;
	sustainLF[621]:=49.400;
	sustainLF[622]:=49.400;
	sustainLF[623]:=49.400;
	sustainLF[624]:=49.400;
	sustainLF[625]:=49.400;
	sustainLF[626]:=49.400;
	sustainLF[627]:=49.400;
	sustainLF[628]:=49.400;
	sustainLF[629]:=49.400;
	sustainLF[630]:=49.400;
	sustainLF[631]:=49.400;
	sustainLF[632]:=49.400;
	sustainLF[633]:=49.400;
	sustainLF[634]:=49.400;
	sustainLF[635]:=49.400;
	sustainLF[636]:=49.400;
	sustainLF[637]:=49.400;
	sustainLF[638]:=49.400;
	sustainLF[639]:=49.400;
	sustainLF[640]:=49.400;
	sustainLF[641]:=49.400;
	sustainLF[642]:=49.400;
	sustainLF[643]:=49.400;
	sustainLF[644]:=49.400;
	sustainLF[645]:=49.400;
	sustainLF[646]:=49.400;
	sustainLF[647]:=49.400;
	sustainLF[648]:=49.400;
	sustainLF[649]:=49.400;
	sustainLF[650]:=49.400;
	sustainLF[651]:=49.400;
	sustainLF[652]:=49.400;
	sustainLF[653]:=49.400;
	sustainLF[654]:=49.400;
	sustainLF[655]:=49.400;
	sustainLF[656]:=49.400;
	sustainLF[657]:=49.400;
	sustainLF[658]:=49.400;
	sustainLF[659]:=49.400;
	sustainLF[660]:=49.400;
	sustainLF[661]:=49.400;
	sustainLF[662]:=49.400;
	sustainLF[663]:=49.400;
	sustainLF[664]:=49.400;
	sustainLF[665]:=49.400;
	sustainLF[666]:=49.400;
	sustainLF[667]:=49.400;
	sustainLF[668]:=49.400;
	sustainLF[669]:=49.400;
	sustainLF[670]:=49.400;
	sustainLF[671]:=49.400;
	sustainLF[672]:=49.400;
	sustainLF[673]:=49.400;
	sustainLF[674]:=49.400;
	sustainLF[675]:=49.400;
	sustainLF[676]:=49.400;
	sustainLF[677]:=49.400;
	sustainLF[678]:=49.400;
	sustainLF[679]:=49.400;
	sustainLF[680]:=49.400;
	sustainLF[681]:=49.400;
	sustainLF[682]:=49.400;
	sustainLF[683]:=49.400;
	sustainLF[684]:=49.400;
	sustainLF[685]:=49.400;
	sustainLF[686]:=49.400;
	sustainLF[687]:=49.400;
	sustainLF[688]:=49.400;
	sustainLF[689]:=49.400;
	sustainLF[690]:=49.400;
	sustainLF[691]:=49.400;
	sustainLF[692]:=49.400;
	sustainLF[693]:=49.400;
	sustainLF[694]:=49.400;
	sustainLF[695]:=49.400;
	sustainLF[696]:=49.400;
	sustainLF[697]:=49.400;
	sustainLF[698]:=49.400;
	sustainLF[699]:=49.400;
	sustainLF[700]:=49.400;
	sustainLF[701]:=49.400;
	sustainLF[702]:=49.400;
	sustainLF[703]:=49.400;
	sustainLF[704]:=49.400;
	sustainLF[705]:=49.400;
	sustainLF[706]:=49.400;
	sustainLF[707]:=49.400;
	sustainLF[708]:=49.400;
	sustainLF[709]:=49.400;
	sustainLF[710]:=49.400;
	sustainLF[711]:=49.400;
	sustainLF[712]:=49.400;
	sustainLF[713]:=49.400;
	sustainLF[714]:=49.400;
	sustainLF[715]:=49.400;
	sustainLF[716]:=49.400;
	sustainLF[717]:=49.400;
	sustainLF[718]:=49.400;
	sustainLF[719]:=49.400;
	sustainLF[720]:=49.400;
	sustainLF[721]:=49.400;
	sustainLF[722]:=49.400;
	sustainLF[723]:=49.400;
	sustainLF[724]:=49.400;
	sustainLF[725]:=49.400;
	sustainLF[726]:=49.400;
	sustainLF[727]:=49.400;
	sustainLF[728]:=49.400;
	sustainLF[729]:=49.400;
	sustainLF[730]:=49.400;
	sustainLF[731]:=49.400;
	sustainLF[732]:=49.400;
	sustainLF[733]:=49.400;
	sustainLF[734]:=49.400;
	sustainLF[735]:=49.400;
	sustainLF[736]:=49.400;
	sustainLF[737]:=49.400;
	sustainLF[738]:=49.400;
	sustainLF[739]:=49.400;
	sustainLF[740]:=49.400;
	sustainLF[741]:=49.400;
	sustainLF[742]:=49.400;
	sustainLF[743]:=49.400;
	sustainLF[744]:=49.400;
	sustainLF[745]:=49.400;
	sustainLF[746]:=49.400;
	sustainLF[747]:=49.400;
	sustainLF[748]:=49.400;
	sustainLF[749]:=49.400;
	sustainLF[750]:=49.400;
	sustainLF[751]:=49.400;
	sustainLF[752]:=49.400;
	sustainLF[753]:=49.400;
	sustainLF[754]:=49.400;
	sustainLF[755]:=49.400;
	sustainLF[756]:=49.400;
	sustainLF[757]:=49.400;
	sustainLF[758]:=49.400;
	sustainLF[759]:=49.400;
	sustainLF[760]:=49.400;
	sustainLF[761]:=49.400;
	sustainLF[762]:=49.400;
	sustainLF[763]:=49.400;
	sustainLF[764]:=49.400;
	sustainLF[765]:=49.400;
	sustainLF[766]:=49.400;
	sustainLF[767]:=49.400;
	sustainLF[768]:=49.400;
	sustainLF[769]:=49.400;
	sustainLF[770]:=49.400;
	sustainLF[771]:=49.400;
	sustainLF[772]:=49.400;
	sustainLF[773]:=49.400;
	sustainLF[774]:=49.400;
	sustainLF[775]:=49.400;
	sustainLF[776]:=49.400;
	sustainLF[777]:=49.400;
	sustainLF[778]:=49.400;
	sustainLF[779]:=49.400;
	sustainLF[780]:=49.400;
	sustainLF[781]:=49.400;
	sustainLF[782]:=49.400;
	sustainLF[783]:=49.400;
	sustainLF[784]:=49.400;
	sustainLF[785]:=49.400;
	sustainLF[786]:=49.400;
	sustainLF[787]:=49.400;
	sustainLF[788]:=49.400;
	sustainLF[789]:=49.400;
	sustainLF[790]:=49.400;
	sustainLF[791]:=49.400;
	sustainLF[792]:=49.400;
	sustainLF[793]:=49.400;
	sustainLF[794]:=49.400;
	sustainLF[795]:=49.400;
	sustainLF[796]:=49.400;
	sustainLF[797]:=49.400;
	sustainLF[798]:=49.400;
	sustainLF[799]:=49.400;
	sustainLF[800]:=49.400;
	sustainLF[801]:=49.400;
	sustainLF[802]:=49.400;
	sustainLF[803]:=49.400;
	sustainLF[804]:=49.400;
	sustainLF[805]:=49.400;
	sustainLF[806]:=49.400;
	sustainLF[807]:=49.400;
	sustainLF[808]:=49.400;
	sustainLF[809]:=49.400;
	sustainLF[810]:=49.400;
	sustainLF[811]:=49.400;
	sustainLF[812]:=49.400;
	sustainLF[813]:=49.400;
	sustainLF[814]:=49.400;
	sustainLF[815]:=49.400;
	sustainLF[816]:=49.400;
	sustainLF[817]:=49.400;
	sustainLF[818]:=49.400;
	sustainLF[819]:=49.400;
	sustainLF[820]:=49.400;
	sustainLF[821]:=49.400;
	sustainLF[822]:=49.400;
	sustainLF[823]:=49.400;
	sustainLF[824]:=49.400;
	sustainLF[825]:=49.400;
	sustainLF[826]:=49.400;
	sustainLF[827]:=49.400;
	sustainLF[828]:=49.400;
	sustainLF[829]:=49.400;
	sustainLF[830]:=49.400;
	sustainLF[831]:=49.400;
	sustainLF[832]:=49.400;
	sustainLF[833]:=49.400;
	sustainLF[834]:=49.400;
	sustainLF[835]:=49.400;
	sustainLF[836]:=49.400;
	sustainLF[837]:=49.400;
	sustainLF[838]:=49.400;
	sustainLF[839]:=49.400;
	sustainLF[840]:=49.400;
	sustainLF[841]:=49.400;
	sustainLF[842]:=49.400;
	sustainLF[843]:=49.400;
	sustainLF[844]:=49.400;
	sustainLF[845]:=49.400;
	sustainLF[846]:=49.400;
	sustainLF[847]:=49.400;
	sustainLF[848]:=49.400;
	sustainLF[849]:=49.400;
	sustainLF[850]:=49.400;
	sustainLF[851]:=49.400;
	sustainLF[852]:=49.400;
	sustainLF[853]:=49.400;
	sustainLF[854]:=49.400;
	sustainLF[855]:=49.400;
	sustainLF[856]:=49.400;
	sustainLF[857]:=49.400;
	sustainLF[858]:=49.400;
	sustainLF[859]:=49.400;
	sustainLF[860]:=49.400;
	sustainLF[861]:=49.400;
	sustainLF[862]:=49.400;
	sustainLF[863]:=49.400;
	sustainLF[864]:=49.400;
	sustainLF[865]:=49.400;
	sustainLF[866]:=49.400;
	sustainLF[867]:=49.400;
	sustainLF[868]:=49.400;
	sustainLF[869]:=49.400;
	sustainLF[870]:=49.400;
	sustainLF[871]:=49.400;
	sustainLF[872]:=49.400;
	sustainLF[873]:=49.400;
	sustainLF[874]:=49.400;
	sustainLF[875]:=49.400;
	sustainLF[876]:=49.400;
	sustainLF[877]:=49.400;
	sustainLF[878]:=49.400;
	sustainLF[879]:=49.400;
	sustainLF[880]:=49.400;
	sustainLF[881]:=49.400;
	sustainLF[882]:=49.400;
	sustainLF[883]:=49.400;
	sustainLF[884]:=49.400;
	sustainLF[885]:=49.400;
	sustainLF[886]:=49.400;
	sustainLF[887]:=49.400;
	sustainLF[888]:=49.400;
	sustainLF[889]:=49.400;
	sustainLF[890]:=49.400;
	sustainLF[891]:=49.400;
	sustainLF[892]:=49.400;
	sustainLF[893]:=49.400;
	sustainLF[894]:=49.400;
	sustainLF[895]:=49.400;
	sustainLF[896]:=49.400;
	sustainLF[897]:=49.400;
	sustainLF[898]:=49.400;
	sustainLF[899]:=49.400;
	sustainLF[900]:=49.400;
	sustainLF[901]:=49.400;
	sustainLF[902]:=49.400;
	sustainLF[903]:=49.400;
	sustainLF[904]:=49.400;
	sustainLF[905]:=49.400;
	sustainLF[906]:=49.400;
	sustainLF[907]:=49.400;
	sustainLF[908]:=49.400;
	sustainLF[909]:=49.400;
	sustainLF[910]:=49.400;
	sustainLF[911]:=49.400;
	sustainLF[912]:=49.400;
	sustainLF[913]:=49.400;
	sustainLF[914]:=49.400;
	sustainLF[915]:=49.400;
	sustainLF[916]:=49.400;
	sustainLF[917]:=49.400;
	sustainLF[918]:=49.400;
	sustainLF[919]:=49.400;
	sustainLF[920]:=49.400;
	sustainLF[921]:=49.400;
	sustainLF[922]:=49.400;
	sustainLF[923]:=49.400;
	sustainLF[924]:=49.400;
	sustainLF[925]:=49.400;
	sustainLF[926]:=49.400;
	sustainLF[927]:=49.400;
	sustainLF[928]:=49.400;
	sustainLF[929]:=49.400;
	sustainLF[930]:=50.000;
	sustainLF[931]:=50.000;
	sustainLF[932]:=50.000;
	sustainLF[933]:=50.000;
	sustainLF[934]:=50.000;
	sustainLF[935]:=50.000;
	sustainLF[936]:=50.000;
	sustainLF[937]:=50.000;
	sustainLF[938]:=50.000;
	sustainLF[939]:=50.000;
	sustainLF[940]:=50.000;
	sustainLF[941]:=50.000;
	sustainLF[942]:=50.000;
	sustainLF[943]:=50.000;
	sustainLF[944]:=50.000;
	sustainLF[945]:=50.000;
	sustainLF[946]:=50.000;
	sustainLF[947]:=50.000;
	sustainLF[948]:=50.000;
	sustainLF[949]:=50.000;
	sustainLF[950]:=50.000;
	sustainLF[951]:=50.000;
	sustainLF[952]:=50.000;
	sustainLF[953]:=50.000;
	sustainLF[954]:=50.000;
	sustainLF[955]:=50.000;
	sustainLF[956]:=50.000;
	sustainLF[957]:=50.000;
	sustainLF[958]:=50.000;
	sustainLF[959]:=50.000;

	stepTestFull[0]:=50.000;
	stepTestFull[1]:=50.000;
	stepTestFull[2]:=50.000;
	stepTestFull[3]:=50.000;
	stepTestFull[4]:=50.000;
	stepTestFull[5]:=50.000;
	stepTestFull[6]:=50.000;
	stepTestFull[7]:=50.000;
	stepTestFull[8]:=50.000;
	stepTestFull[9]:=50.000;
	stepTestFull[10]:=50.000;
	stepTestFull[11]:=50.000;
	stepTestFull[12]:=50.000;
	stepTestFull[13]:=50.000;
	stepTestFull[14]:=50.000;
	stepTestFull[15]:=50.000;
	stepTestFull[16]:=50.000;
	stepTestFull[17]:=50.000;
	stepTestFull[18]:=50.000;
	stepTestFull[19]:=50.000;
	stepTestFull[20]:=50.000;
	stepTestFull[21]:=50.000;
	stepTestFull[22]:=50.000;
	stepTestFull[23]:=50.000;
	stepTestFull[24]:=50.000;
	stepTestFull[25]:=50.000;
	stepTestFull[26]:=50.000;
	stepTestFull[27]:=50.000;
	stepTestFull[28]:=50.000;
	stepTestFull[29]:=50.000;
	stepTestFull[30]:=50.010;
	stepTestFull[31]:=50.010;
	stepTestFull[32]:=50.010;
	stepTestFull[33]:=50.010;
	stepTestFull[34]:=50.010;
	stepTestFull[35]:=50.010;
	stepTestFull[36]:=50.010;
	stepTestFull[37]:=50.010;
	stepTestFull[38]:=50.010;
	stepTestFull[39]:=50.010;
	stepTestFull[40]:=50.010;
	stepTestFull[41]:=50.010;
	stepTestFull[42]:=50.010;
	stepTestFull[43]:=50.010;
	stepTestFull[44]:=50.010;
	stepTestFull[45]:=50.010;
	stepTestFull[46]:=50.010;
	stepTestFull[47]:=50.010;
	stepTestFull[48]:=50.010;
	stepTestFull[49]:=50.010;
	stepTestFull[50]:=50.010;
	stepTestFull[51]:=50.010;
	stepTestFull[52]:=50.010;
	stepTestFull[53]:=50.010;
	stepTestFull[54]:=50.010;
	stepTestFull[55]:=50.010;
	stepTestFull[56]:=50.010;
	stepTestFull[57]:=50.010;
	stepTestFull[58]:=50.010;
	stepTestFull[59]:=50.010;
	stepTestFull[60]:=50.010;
	stepTestFull[61]:=50.010;
	stepTestFull[62]:=50.010;
	stepTestFull[63]:=50.010;
	stepTestFull[64]:=50.010;
	stepTestFull[65]:=50.010;
	stepTestFull[66]:=50.010;
	stepTestFull[67]:=50.010;
	stepTestFull[68]:=50.010;
	stepTestFull[69]:=50.010;
	stepTestFull[70]:=50.010;
	stepTestFull[71]:=50.010;
	stepTestFull[72]:=50.010;
	stepTestFull[73]:=50.010;
	stepTestFull[74]:=50.010;
	stepTestFull[75]:=50.010;
	stepTestFull[76]:=50.010;
	stepTestFull[77]:=50.010;
	stepTestFull[78]:=50.010;
	stepTestFull[79]:=50.010;
	stepTestFull[80]:=50.010;
	stepTestFull[81]:=50.010;
	stepTestFull[82]:=50.010;
	stepTestFull[83]:=50.010;
	stepTestFull[84]:=50.010;
	stepTestFull[85]:=50.010;
	stepTestFull[86]:=50.010;
	stepTestFull[87]:=50.010;
	stepTestFull[88]:=50.010;
	stepTestFull[89]:=50.010;
	stepTestFull[90]:=50.010;
	stepTestFull[91]:=50.010;
	stepTestFull[92]:=50.010;
	stepTestFull[93]:=50.010;
	stepTestFull[94]:=50.010;
	stepTestFull[95]:=50.010;
	stepTestFull[96]:=50.010;
	stepTestFull[97]:=50.010;
	stepTestFull[98]:=50.010;
	stepTestFull[99]:=50.010;
	stepTestFull[100]:=50.010;
	stepTestFull[101]:=50.010;
	stepTestFull[102]:=50.010;
	stepTestFull[103]:=50.010;
	stepTestFull[104]:=50.010;
	stepTestFull[105]:=50.010;
	stepTestFull[106]:=50.010;
	stepTestFull[107]:=50.010;
	stepTestFull[108]:=50.010;
	stepTestFull[109]:=50.010;
	stepTestFull[110]:=50.010;
	stepTestFull[111]:=50.010;
	stepTestFull[112]:=50.010;
	stepTestFull[113]:=50.010;
	stepTestFull[114]:=50.010;
	stepTestFull[115]:=50.010;
	stepTestFull[116]:=50.010;
	stepTestFull[117]:=50.010;
	stepTestFull[118]:=50.010;
	stepTestFull[119]:=50.010;
	stepTestFull[120]:=50.010;
	stepTestFull[121]:=50.010;
	stepTestFull[122]:=50.010;
	stepTestFull[123]:=50.010;
	stepTestFull[124]:=50.010;
	stepTestFull[125]:=50.010;
	stepTestFull[126]:=50.010;
	stepTestFull[127]:=50.010;
	stepTestFull[128]:=50.010;
	stepTestFull[129]:=50.010;
	stepTestFull[130]:=50.010;
	stepTestFull[131]:=50.010;
	stepTestFull[132]:=50.010;
	stepTestFull[133]:=50.010;
	stepTestFull[134]:=50.010;
	stepTestFull[135]:=50.010;
	stepTestFull[136]:=50.010;
	stepTestFull[137]:=50.010;
	stepTestFull[138]:=50.010;
	stepTestFull[139]:=50.010;
	stepTestFull[140]:=50.010;
	stepTestFull[141]:=50.010;
	stepTestFull[142]:=50.010;
	stepTestFull[143]:=50.010;
	stepTestFull[144]:=50.010;
	stepTestFull[145]:=50.010;
	stepTestFull[146]:=50.010;
	stepTestFull[147]:=50.010;
	stepTestFull[148]:=50.010;
	stepTestFull[149]:=50.010;
	stepTestFull[150]:=50.010;
	stepTestFull[151]:=50.010;
	stepTestFull[152]:=50.010;
	stepTestFull[153]:=50.010;
	stepTestFull[154]:=50.010;
	stepTestFull[155]:=50.010;
	stepTestFull[156]:=50.010;
	stepTestFull[157]:=50.010;
	stepTestFull[158]:=50.010;
	stepTestFull[159]:=50.010;
	stepTestFull[160]:=50.010;
	stepTestFull[161]:=50.010;
	stepTestFull[162]:=50.010;
	stepTestFull[163]:=50.010;
	stepTestFull[164]:=50.010;
	stepTestFull[165]:=50.010;
	stepTestFull[166]:=50.010;
	stepTestFull[167]:=50.010;
	stepTestFull[168]:=50.010;
	stepTestFull[169]:=50.010;
	stepTestFull[170]:=50.010;
	stepTestFull[171]:=50.010;
	stepTestFull[172]:=50.010;
	stepTestFull[173]:=50.010;
	stepTestFull[174]:=50.010;
	stepTestFull[175]:=50.010;
	stepTestFull[176]:=50.010;
	stepTestFull[177]:=50.010;
	stepTestFull[178]:=50.010;
	stepTestFull[179]:=50.010;
	stepTestFull[180]:=50.010;
	stepTestFull[181]:=50.010;
	stepTestFull[182]:=50.010;
	stepTestFull[183]:=50.010;
	stepTestFull[184]:=50.010;
	stepTestFull[185]:=50.010;
	stepTestFull[186]:=50.010;
	stepTestFull[187]:=50.010;
	stepTestFull[188]:=50.010;
	stepTestFull[189]:=50.010;
	stepTestFull[190]:=50.010;
	stepTestFull[191]:=50.010;
	stepTestFull[192]:=50.010;
	stepTestFull[193]:=50.010;
	stepTestFull[194]:=50.010;
	stepTestFull[195]:=50.010;
	stepTestFull[196]:=50.010;
	stepTestFull[197]:=50.010;
	stepTestFull[198]:=50.010;
	stepTestFull[199]:=50.010;
	stepTestFull[200]:=50.010;
	stepTestFull[201]:=50.010;
	stepTestFull[202]:=50.010;
	stepTestFull[203]:=50.010;
	stepTestFull[204]:=50.010;
	stepTestFull[205]:=50.010;
	stepTestFull[206]:=50.010;
	stepTestFull[207]:=50.010;
	stepTestFull[208]:=50.010;
	stepTestFull[209]:=50.010;
	stepTestFull[210]:=50.000;
	stepTestFull[211]:=50.000;
	stepTestFull[212]:=50.000;
	stepTestFull[213]:=50.000;
	stepTestFull[214]:=50.000;
	stepTestFull[215]:=50.000;
	stepTestFull[216]:=50.000;
	stepTestFull[217]:=50.000;
	stepTestFull[218]:=50.000;
	stepTestFull[219]:=50.000;
	stepTestFull[220]:=50.000;
	stepTestFull[221]:=50.000;
	stepTestFull[222]:=50.000;
	stepTestFull[223]:=50.000;
	stepTestFull[224]:=50.000;
	stepTestFull[225]:=50.000;
	stepTestFull[226]:=50.000;
	stepTestFull[227]:=50.000;
	stepTestFull[228]:=50.000;
	stepTestFull[229]:=50.000;
	stepTestFull[230]:=50.000;
	stepTestFull[231]:=50.000;
	stepTestFull[232]:=50.000;
	stepTestFull[233]:=50.000;
	stepTestFull[234]:=50.000;
	stepTestFull[235]:=50.000;
	stepTestFull[236]:=50.000;
	stepTestFull[237]:=50.000;
	stepTestFull[238]:=50.000;
	stepTestFull[239]:=50.000;
	stepTestFull[240]:=50.000;
	stepTestFull[241]:=50.000;
	stepTestFull[242]:=50.000;
	stepTestFull[243]:=50.000;
	stepTestFull[244]:=50.000;
	stepTestFull[245]:=50.000;
	stepTestFull[246]:=50.000;
	stepTestFull[247]:=50.000;
	stepTestFull[248]:=50.000;
	stepTestFull[249]:=50.000;
	stepTestFull[250]:=50.000;
	stepTestFull[251]:=50.000;
	stepTestFull[252]:=50.000;
	stepTestFull[253]:=50.000;
	stepTestFull[254]:=50.000;
	stepTestFull[255]:=50.000;
	stepTestFull[256]:=50.000;
	stepTestFull[257]:=50.000;
	stepTestFull[258]:=50.000;
	stepTestFull[259]:=50.000;
	stepTestFull[260]:=50.000;
	stepTestFull[261]:=50.000;
	stepTestFull[262]:=50.000;
	stepTestFull[263]:=50.000;
	stepTestFull[264]:=50.000;
	stepTestFull[265]:=50.000;
	stepTestFull[266]:=50.000;
	stepTestFull[267]:=50.000;
	stepTestFull[268]:=50.000;
	stepTestFull[269]:=50.000;
	stepTestFull[270]:=49.990;
	stepTestFull[271]:=49.990;
	stepTestFull[272]:=49.990;
	stepTestFull[273]:=49.990;
	stepTestFull[274]:=49.990;
	stepTestFull[275]:=49.990;
	stepTestFull[276]:=49.990;
	stepTestFull[277]:=49.990;
	stepTestFull[278]:=49.990;
	stepTestFull[279]:=49.990;
	stepTestFull[280]:=49.990;
	stepTestFull[281]:=49.990;
	stepTestFull[282]:=49.990;
	stepTestFull[283]:=49.990;
	stepTestFull[284]:=49.990;
	stepTestFull[285]:=49.990;
	stepTestFull[286]:=49.990;
	stepTestFull[287]:=49.990;
	stepTestFull[288]:=49.990;
	stepTestFull[289]:=49.990;
	stepTestFull[290]:=49.990;
	stepTestFull[291]:=49.990;
	stepTestFull[292]:=49.990;
	stepTestFull[293]:=49.990;
	stepTestFull[294]:=49.990;
	stepTestFull[295]:=49.990;
	stepTestFull[296]:=49.990;
	stepTestFull[297]:=49.990;
	stepTestFull[298]:=49.990;
	stepTestFull[299]:=49.990;
	stepTestFull[300]:=49.990;
	stepTestFull[301]:=49.990;
	stepTestFull[302]:=49.990;
	stepTestFull[303]:=49.990;
	stepTestFull[304]:=49.990;
	stepTestFull[305]:=49.990;
	stepTestFull[306]:=49.990;
	stepTestFull[307]:=49.990;
	stepTestFull[308]:=49.990;
	stepTestFull[309]:=49.990;
	stepTestFull[310]:=49.990;
	stepTestFull[311]:=49.990;
	stepTestFull[312]:=49.990;
	stepTestFull[313]:=49.990;
	stepTestFull[314]:=49.990;
	stepTestFull[315]:=49.990;
	stepTestFull[316]:=49.990;
	stepTestFull[317]:=49.990;
	stepTestFull[318]:=49.990;
	stepTestFull[319]:=49.990;
	stepTestFull[320]:=49.990;
	stepTestFull[321]:=49.990;
	stepTestFull[322]:=49.990;
	stepTestFull[323]:=49.990;
	stepTestFull[324]:=49.990;
	stepTestFull[325]:=49.990;
	stepTestFull[326]:=49.990;
	stepTestFull[327]:=49.990;
	stepTestFull[328]:=49.990;
	stepTestFull[329]:=49.990;
	stepTestFull[330]:=49.990;
	stepTestFull[331]:=49.990;
	stepTestFull[332]:=49.990;
	stepTestFull[333]:=49.990;
	stepTestFull[334]:=49.990;
	stepTestFull[335]:=49.990;
	stepTestFull[336]:=49.990;
	stepTestFull[337]:=49.990;
	stepTestFull[338]:=49.990;
	stepTestFull[339]:=49.990;
	stepTestFull[340]:=49.990;
	stepTestFull[341]:=49.990;
	stepTestFull[342]:=49.990;
	stepTestFull[343]:=49.990;
	stepTestFull[344]:=49.990;
	stepTestFull[345]:=49.990;
	stepTestFull[346]:=49.990;
	stepTestFull[347]:=49.990;
	stepTestFull[348]:=49.990;
	stepTestFull[349]:=49.990;
	stepTestFull[350]:=49.990;
	stepTestFull[351]:=49.990;
	stepTestFull[352]:=49.990;
	stepTestFull[353]:=49.990;
	stepTestFull[354]:=49.990;
	stepTestFull[355]:=49.990;
	stepTestFull[356]:=49.990;
	stepTestFull[357]:=49.990;
	stepTestFull[358]:=49.990;
	stepTestFull[359]:=49.990;
	stepTestFull[360]:=49.990;
	stepTestFull[361]:=49.990;
	stepTestFull[362]:=49.990;
	stepTestFull[363]:=49.990;
	stepTestFull[364]:=49.990;
	stepTestFull[365]:=49.990;
	stepTestFull[366]:=49.990;
	stepTestFull[367]:=49.990;
	stepTestFull[368]:=49.990;
	stepTestFull[369]:=49.990;
	stepTestFull[370]:=49.990;
	stepTestFull[371]:=49.990;
	stepTestFull[372]:=49.990;
	stepTestFull[373]:=49.990;
	stepTestFull[374]:=49.990;
	stepTestFull[375]:=49.990;
	stepTestFull[376]:=49.990;
	stepTestFull[377]:=49.990;
	stepTestFull[378]:=49.990;
	stepTestFull[379]:=49.990;
	stepTestFull[380]:=49.990;
	stepTestFull[381]:=49.990;
	stepTestFull[382]:=49.990;
	stepTestFull[383]:=49.990;
	stepTestFull[384]:=49.990;
	stepTestFull[385]:=49.990;
	stepTestFull[386]:=49.990;
	stepTestFull[387]:=49.990;
	stepTestFull[388]:=49.990;
	stepTestFull[389]:=49.990;
	stepTestFull[390]:=49.990;
	stepTestFull[391]:=49.990;
	stepTestFull[392]:=49.990;
	stepTestFull[393]:=49.990;
	stepTestFull[394]:=49.990;
	stepTestFull[395]:=49.990;
	stepTestFull[396]:=49.990;
	stepTestFull[397]:=49.990;
	stepTestFull[398]:=49.990;
	stepTestFull[399]:=49.990;
	stepTestFull[400]:=49.990;
	stepTestFull[401]:=49.990;
	stepTestFull[402]:=49.990;
	stepTestFull[403]:=49.990;
	stepTestFull[404]:=49.990;
	stepTestFull[405]:=49.990;
	stepTestFull[406]:=49.990;
	stepTestFull[407]:=49.990;
	stepTestFull[408]:=49.990;
	stepTestFull[409]:=49.990;
	stepTestFull[410]:=49.990;
	stepTestFull[411]:=49.990;
	stepTestFull[412]:=49.990;
	stepTestFull[413]:=49.990;
	stepTestFull[414]:=49.990;
	stepTestFull[415]:=49.990;
	stepTestFull[416]:=49.990;
	stepTestFull[417]:=49.990;
	stepTestFull[418]:=49.990;
	stepTestFull[419]:=49.990;
	stepTestFull[420]:=49.990;
	stepTestFull[421]:=49.990;
	stepTestFull[422]:=49.990;
	stepTestFull[423]:=49.990;
	stepTestFull[424]:=49.990;
	stepTestFull[425]:=49.990;
	stepTestFull[426]:=49.990;
	stepTestFull[427]:=49.990;
	stepTestFull[428]:=49.990;
	stepTestFull[429]:=49.990;
	stepTestFull[430]:=49.990;
	stepTestFull[431]:=49.990;
	stepTestFull[432]:=49.990;
	stepTestFull[433]:=49.990;
	stepTestFull[434]:=49.990;
	stepTestFull[435]:=49.990;
	stepTestFull[436]:=49.990;
	stepTestFull[437]:=49.990;
	stepTestFull[438]:=49.990;
	stepTestFull[439]:=49.990;
	stepTestFull[440]:=49.990;
	stepTestFull[441]:=49.990;
	stepTestFull[442]:=49.990;
	stepTestFull[443]:=49.990;
	stepTestFull[444]:=49.990;
	stepTestFull[445]:=49.990;
	stepTestFull[446]:=49.990;
	stepTestFull[447]:=49.990;
	stepTestFull[448]:=49.990;
	stepTestFull[449]:=49.990;
	stepTestFull[450]:=50.000;
	stepTestFull[451]:=50.000;
	stepTestFull[452]:=50.000;
	stepTestFull[453]:=50.000;
	stepTestFull[454]:=50.000;
	stepTestFull[455]:=50.000;
	stepTestFull[456]:=50.000;
	stepTestFull[457]:=50.000;
	stepTestFull[458]:=50.000;
	stepTestFull[459]:=50.000;
	stepTestFull[460]:=50.000;
	stepTestFull[461]:=50.000;
	stepTestFull[462]:=50.000;
	stepTestFull[463]:=50.000;
	stepTestFull[464]:=50.000;
	stepTestFull[465]:=50.000;
	stepTestFull[466]:=50.000;
	stepTestFull[467]:=50.000;
	stepTestFull[468]:=50.000;
	stepTestFull[469]:=50.000;
	stepTestFull[470]:=50.000;
	stepTestFull[471]:=50.000;
	stepTestFull[472]:=50.000;
	stepTestFull[473]:=50.000;
	stepTestFull[474]:=50.000;
	stepTestFull[475]:=50.000;
	stepTestFull[476]:=50.000;
	stepTestFull[477]:=50.000;
	stepTestFull[478]:=50.000;
	stepTestFull[479]:=50.000;
	stepTestFull[480]:=50.000;
	stepTestFull[481]:=50.000;
	stepTestFull[482]:=50.000;
	stepTestFull[483]:=50.000;
	stepTestFull[484]:=50.000;
	stepTestFull[485]:=50.000;
	stepTestFull[486]:=50.000;
	stepTestFull[487]:=50.000;
	stepTestFull[488]:=50.000;
	stepTestFull[489]:=50.000;
	stepTestFull[490]:=50.000;
	stepTestFull[491]:=50.000;
	stepTestFull[492]:=50.000;
	stepTestFull[493]:=50.000;
	stepTestFull[494]:=50.000;
	stepTestFull[495]:=50.000;
	stepTestFull[496]:=50.000;
	stepTestFull[497]:=50.000;
	stepTestFull[498]:=50.000;
	stepTestFull[499]:=50.000;
	stepTestFull[500]:=50.000;
	stepTestFull[501]:=50.000;
	stepTestFull[502]:=50.000;
	stepTestFull[503]:=50.000;
	stepTestFull[504]:=50.000;
	stepTestFull[505]:=50.000;
	stepTestFull[506]:=50.000;
	stepTestFull[507]:=50.000;
	stepTestFull[508]:=50.000;
	stepTestFull[509]:=50.000;
	stepTestFull[510]:=50.020;
	stepTestFull[511]:=50.020;
	stepTestFull[512]:=50.020;
	stepTestFull[513]:=50.020;
	stepTestFull[514]:=50.020;
	stepTestFull[515]:=50.020;
	stepTestFull[516]:=50.020;
	stepTestFull[517]:=50.020;
	stepTestFull[518]:=50.020;
	stepTestFull[519]:=50.020;
	stepTestFull[520]:=50.020;
	stepTestFull[521]:=50.020;
	stepTestFull[522]:=50.020;
	stepTestFull[523]:=50.020;
	stepTestFull[524]:=50.020;
	stepTestFull[525]:=50.020;
	stepTestFull[526]:=50.020;
	stepTestFull[527]:=50.020;
	stepTestFull[528]:=50.020;
	stepTestFull[529]:=50.020;
	stepTestFull[530]:=50.020;
	stepTestFull[531]:=50.020;
	stepTestFull[532]:=50.020;
	stepTestFull[533]:=50.020;
	stepTestFull[534]:=50.020;
	stepTestFull[535]:=50.020;
	stepTestFull[536]:=50.020;
	stepTestFull[537]:=50.020;
	stepTestFull[538]:=50.020;
	stepTestFull[539]:=50.020;
	stepTestFull[540]:=50.020;
	stepTestFull[541]:=50.020;
	stepTestFull[542]:=50.020;
	stepTestFull[543]:=50.020;
	stepTestFull[544]:=50.020;
	stepTestFull[545]:=50.020;
	stepTestFull[546]:=50.020;
	stepTestFull[547]:=50.020;
	stepTestFull[548]:=50.020;
	stepTestFull[549]:=50.020;
	stepTestFull[550]:=50.020;
	stepTestFull[551]:=50.020;
	stepTestFull[552]:=50.020;
	stepTestFull[553]:=50.020;
	stepTestFull[554]:=50.020;
	stepTestFull[555]:=50.020;
	stepTestFull[556]:=50.020;
	stepTestFull[557]:=50.020;
	stepTestFull[558]:=50.020;
	stepTestFull[559]:=50.020;
	stepTestFull[560]:=50.020;
	stepTestFull[561]:=50.020;
	stepTestFull[562]:=50.020;
	stepTestFull[563]:=50.020;
	stepTestFull[564]:=50.020;
	stepTestFull[565]:=50.020;
	stepTestFull[566]:=50.020;
	stepTestFull[567]:=50.020;
	stepTestFull[568]:=50.020;
	stepTestFull[569]:=50.020;
	stepTestFull[570]:=50.020;
	stepTestFull[571]:=50.020;
	stepTestFull[572]:=50.020;
	stepTestFull[573]:=50.020;
	stepTestFull[574]:=50.020;
	stepTestFull[575]:=50.020;
	stepTestFull[576]:=50.020;
	stepTestFull[577]:=50.020;
	stepTestFull[578]:=50.020;
	stepTestFull[579]:=50.020;
	stepTestFull[580]:=50.020;
	stepTestFull[581]:=50.020;
	stepTestFull[582]:=50.020;
	stepTestFull[583]:=50.020;
	stepTestFull[584]:=50.020;
	stepTestFull[585]:=50.020;
	stepTestFull[586]:=50.020;
	stepTestFull[587]:=50.020;
	stepTestFull[588]:=50.020;
	stepTestFull[589]:=50.020;
	stepTestFull[590]:=50.020;
	stepTestFull[591]:=50.020;
	stepTestFull[592]:=50.020;
	stepTestFull[593]:=50.020;
	stepTestFull[594]:=50.020;
	stepTestFull[595]:=50.020;
	stepTestFull[596]:=50.020;
	stepTestFull[597]:=50.020;
	stepTestFull[598]:=50.020;
	stepTestFull[599]:=50.020;
	stepTestFull[600]:=50.020;
	stepTestFull[601]:=50.020;
	stepTestFull[602]:=50.020;
	stepTestFull[603]:=50.020;
	stepTestFull[604]:=50.020;
	stepTestFull[605]:=50.020;
	stepTestFull[606]:=50.020;
	stepTestFull[607]:=50.020;
	stepTestFull[608]:=50.020;
	stepTestFull[609]:=50.020;
	stepTestFull[610]:=50.020;
	stepTestFull[611]:=50.020;
	stepTestFull[612]:=50.020;
	stepTestFull[613]:=50.020;
	stepTestFull[614]:=50.020;
	stepTestFull[615]:=50.020;
	stepTestFull[616]:=50.020;
	stepTestFull[617]:=50.020;
	stepTestFull[618]:=50.020;
	stepTestFull[619]:=50.020;
	stepTestFull[620]:=50.020;
	stepTestFull[621]:=50.020;
	stepTestFull[622]:=50.020;
	stepTestFull[623]:=50.020;
	stepTestFull[624]:=50.020;
	stepTestFull[625]:=50.020;
	stepTestFull[626]:=50.020;
	stepTestFull[627]:=50.020;
	stepTestFull[628]:=50.020;
	stepTestFull[629]:=50.020;
	stepTestFull[630]:=50.020;
	stepTestFull[631]:=50.020;
	stepTestFull[632]:=50.020;
	stepTestFull[633]:=50.020;
	stepTestFull[634]:=50.020;
	stepTestFull[635]:=50.020;
	stepTestFull[636]:=50.020;
	stepTestFull[637]:=50.020;
	stepTestFull[638]:=50.020;
	stepTestFull[639]:=50.020;
	stepTestFull[640]:=50.020;
	stepTestFull[641]:=50.020;
	stepTestFull[642]:=50.020;
	stepTestFull[643]:=50.020;
	stepTestFull[644]:=50.020;
	stepTestFull[645]:=50.020;
	stepTestFull[646]:=50.020;
	stepTestFull[647]:=50.020;
	stepTestFull[648]:=50.020;
	stepTestFull[649]:=50.020;
	stepTestFull[650]:=50.020;
	stepTestFull[651]:=50.020;
	stepTestFull[652]:=50.020;
	stepTestFull[653]:=50.020;
	stepTestFull[654]:=50.020;
	stepTestFull[655]:=50.020;
	stepTestFull[656]:=50.020;
	stepTestFull[657]:=50.020;
	stepTestFull[658]:=50.020;
	stepTestFull[659]:=50.020;
	stepTestFull[660]:=50.020;
	stepTestFull[661]:=50.020;
	stepTestFull[662]:=50.020;
	stepTestFull[663]:=50.020;
	stepTestFull[664]:=50.020;
	stepTestFull[665]:=50.020;
	stepTestFull[666]:=50.020;
	stepTestFull[667]:=50.020;
	stepTestFull[668]:=50.020;
	stepTestFull[669]:=50.020;
	stepTestFull[670]:=50.020;
	stepTestFull[671]:=50.020;
	stepTestFull[672]:=50.020;
	stepTestFull[673]:=50.020;
	stepTestFull[674]:=50.020;
	stepTestFull[675]:=50.020;
	stepTestFull[676]:=50.020;
	stepTestFull[677]:=50.020;
	stepTestFull[678]:=50.020;
	stepTestFull[679]:=50.020;
	stepTestFull[680]:=50.020;
	stepTestFull[681]:=50.020;
	stepTestFull[682]:=50.020;
	stepTestFull[683]:=50.020;
	stepTestFull[684]:=50.020;
	stepTestFull[685]:=50.020;
	stepTestFull[686]:=50.020;
	stepTestFull[687]:=50.020;
	stepTestFull[688]:=50.020;
	stepTestFull[689]:=50.020;
	stepTestFull[690]:=50.000;
	stepTestFull[691]:=50.000;
	stepTestFull[692]:=50.000;
	stepTestFull[693]:=50.000;
	stepTestFull[694]:=50.000;
	stepTestFull[695]:=50.000;
	stepTestFull[696]:=50.000;
	stepTestFull[697]:=50.000;
	stepTestFull[698]:=50.000;
	stepTestFull[699]:=50.000;
	stepTestFull[700]:=50.000;
	stepTestFull[701]:=50.000;
	stepTestFull[702]:=50.000;
	stepTestFull[703]:=50.000;
	stepTestFull[704]:=50.000;
	stepTestFull[705]:=50.000;
	stepTestFull[706]:=50.000;
	stepTestFull[707]:=50.000;
	stepTestFull[708]:=50.000;
	stepTestFull[709]:=50.000;
	stepTestFull[710]:=50.000;
	stepTestFull[711]:=50.000;
	stepTestFull[712]:=50.000;
	stepTestFull[713]:=50.000;
	stepTestFull[714]:=50.000;
	stepTestFull[715]:=50.000;
	stepTestFull[716]:=50.000;
	stepTestFull[717]:=50.000;
	stepTestFull[718]:=50.000;
	stepTestFull[719]:=50.000;
	stepTestFull[720]:=50.000;
	stepTestFull[721]:=50.000;
	stepTestFull[722]:=50.000;
	stepTestFull[723]:=50.000;
	stepTestFull[724]:=50.000;
	stepTestFull[725]:=50.000;
	stepTestFull[726]:=50.000;
	stepTestFull[727]:=50.000;
	stepTestFull[728]:=50.000;
	stepTestFull[729]:=50.000;
	stepTestFull[730]:=50.000;
	stepTestFull[731]:=50.000;
	stepTestFull[732]:=50.000;
	stepTestFull[733]:=50.000;
	stepTestFull[734]:=50.000;
	stepTestFull[735]:=50.000;
	stepTestFull[736]:=50.000;
	stepTestFull[737]:=50.000;
	stepTestFull[738]:=50.000;
	stepTestFull[739]:=50.000;
	stepTestFull[740]:=50.000;
	stepTestFull[741]:=50.000;
	stepTestFull[742]:=50.000;
	stepTestFull[743]:=50.000;
	stepTestFull[744]:=50.000;
	stepTestFull[745]:=50.000;
	stepTestFull[746]:=50.000;
	stepTestFull[747]:=50.000;
	stepTestFull[748]:=50.000;
	stepTestFull[749]:=50.000;
	stepTestFull[750]:=49.980;
	stepTestFull[751]:=49.980;
	stepTestFull[752]:=49.980;
	stepTestFull[753]:=49.980;
	stepTestFull[754]:=49.980;
	stepTestFull[755]:=49.980;
	stepTestFull[756]:=49.980;
	stepTestFull[757]:=49.980;
	stepTestFull[758]:=49.980;
	stepTestFull[759]:=49.980;
	stepTestFull[760]:=49.980;
	stepTestFull[761]:=49.980;
	stepTestFull[762]:=49.980;
	stepTestFull[763]:=49.980;
	stepTestFull[764]:=49.980;
	stepTestFull[765]:=49.980;
	stepTestFull[766]:=49.980;
	stepTestFull[767]:=49.980;
	stepTestFull[768]:=49.980;
	stepTestFull[769]:=49.980;
	stepTestFull[770]:=49.980;
	stepTestFull[771]:=49.980;
	stepTestFull[772]:=49.980;
	stepTestFull[773]:=49.980;
	stepTestFull[774]:=49.980;
	stepTestFull[775]:=49.980;
	stepTestFull[776]:=49.980;
	stepTestFull[777]:=49.980;
	stepTestFull[778]:=49.980;
	stepTestFull[779]:=49.980;
	stepTestFull[780]:=49.980;
	stepTestFull[781]:=49.980;
	stepTestFull[782]:=49.980;
	stepTestFull[783]:=49.980;
	stepTestFull[784]:=49.980;
	stepTestFull[785]:=49.980;
	stepTestFull[786]:=49.980;
	stepTestFull[787]:=49.980;
	stepTestFull[788]:=49.980;
	stepTestFull[789]:=49.980;
	stepTestFull[790]:=49.980;
	stepTestFull[791]:=49.980;
	stepTestFull[792]:=49.980;
	stepTestFull[793]:=49.980;
	stepTestFull[794]:=49.980;
	stepTestFull[795]:=49.980;
	stepTestFull[796]:=49.980;
	stepTestFull[797]:=49.980;
	stepTestFull[798]:=49.980;
	stepTestFull[799]:=49.980;
	stepTestFull[800]:=49.980;
	stepTestFull[801]:=49.980;
	stepTestFull[802]:=49.980;
	stepTestFull[803]:=49.980;
	stepTestFull[804]:=49.980;
	stepTestFull[805]:=49.980;
	stepTestFull[806]:=49.980;
	stepTestFull[807]:=49.980;
	stepTestFull[808]:=49.980;
	stepTestFull[809]:=49.980;
	stepTestFull[810]:=49.980;
	stepTestFull[811]:=49.980;
	stepTestFull[812]:=49.980;
	stepTestFull[813]:=49.980;
	stepTestFull[814]:=49.980;
	stepTestFull[815]:=49.980;
	stepTestFull[816]:=49.980;
	stepTestFull[817]:=49.980;
	stepTestFull[818]:=49.980;
	stepTestFull[819]:=49.980;
	stepTestFull[820]:=49.980;
	stepTestFull[821]:=49.980;
	stepTestFull[822]:=49.980;
	stepTestFull[823]:=49.980;
	stepTestFull[824]:=49.980;
	stepTestFull[825]:=49.980;
	stepTestFull[826]:=49.980;
	stepTestFull[827]:=49.980;
	stepTestFull[828]:=49.980;
	stepTestFull[829]:=49.980;
	stepTestFull[830]:=49.980;
	stepTestFull[831]:=49.980;
	stepTestFull[832]:=49.980;
	stepTestFull[833]:=49.980;
	stepTestFull[834]:=49.980;
	stepTestFull[835]:=49.980;
	stepTestFull[836]:=49.980;
	stepTestFull[837]:=49.980;
	stepTestFull[838]:=49.980;
	stepTestFull[839]:=49.980;
	stepTestFull[840]:=49.980;
	stepTestFull[841]:=49.980;
	stepTestFull[842]:=49.980;
	stepTestFull[843]:=49.980;
	stepTestFull[844]:=49.980;
	stepTestFull[845]:=49.980;
	stepTestFull[846]:=49.980;
	stepTestFull[847]:=49.980;
	stepTestFull[848]:=49.980;
	stepTestFull[849]:=49.980;
	stepTestFull[850]:=49.980;
	stepTestFull[851]:=49.980;
	stepTestFull[852]:=49.980;
	stepTestFull[853]:=49.980;
	stepTestFull[854]:=49.980;
	stepTestFull[855]:=49.980;
	stepTestFull[856]:=49.980;
	stepTestFull[857]:=49.980;
	stepTestFull[858]:=49.980;
	stepTestFull[859]:=49.980;
	stepTestFull[860]:=49.980;
	stepTestFull[861]:=49.980;
	stepTestFull[862]:=49.980;
	stepTestFull[863]:=49.980;
	stepTestFull[864]:=49.980;
	stepTestFull[865]:=49.980;
	stepTestFull[866]:=49.980;
	stepTestFull[867]:=49.980;
	stepTestFull[868]:=49.980;
	stepTestFull[869]:=49.980;
	stepTestFull[870]:=49.980;
	stepTestFull[871]:=49.980;
	stepTestFull[872]:=49.980;
	stepTestFull[873]:=49.980;
	stepTestFull[874]:=49.980;
	stepTestFull[875]:=49.980;
	stepTestFull[876]:=49.980;
	stepTestFull[877]:=49.980;
	stepTestFull[878]:=49.980;
	stepTestFull[879]:=49.980;
	stepTestFull[880]:=49.980;
	stepTestFull[881]:=49.980;
	stepTestFull[882]:=49.980;
	stepTestFull[883]:=49.980;
	stepTestFull[884]:=49.980;
	stepTestFull[885]:=49.980;
	stepTestFull[886]:=49.980;
	stepTestFull[887]:=49.980;
	stepTestFull[888]:=49.980;
	stepTestFull[889]:=49.980;
	stepTestFull[890]:=49.980;
	stepTestFull[891]:=49.980;
	stepTestFull[892]:=49.980;
	stepTestFull[893]:=49.980;
	stepTestFull[894]:=49.980;
	stepTestFull[895]:=49.980;
	stepTestFull[896]:=49.980;
	stepTestFull[897]:=49.980;
	stepTestFull[898]:=49.980;
	stepTestFull[899]:=49.980;
	stepTestFull[900]:=49.980;
	stepTestFull[901]:=49.980;
	stepTestFull[902]:=49.980;
	stepTestFull[903]:=49.980;
	stepTestFull[904]:=49.980;
	stepTestFull[905]:=49.980;
	stepTestFull[906]:=49.980;
	stepTestFull[907]:=49.980;
	stepTestFull[908]:=49.980;
	stepTestFull[909]:=49.980;
	stepTestFull[910]:=49.980;
	stepTestFull[911]:=49.980;
	stepTestFull[912]:=49.980;
	stepTestFull[913]:=49.980;
	stepTestFull[914]:=49.980;
	stepTestFull[915]:=49.980;
	stepTestFull[916]:=49.980;
	stepTestFull[917]:=49.980;
	stepTestFull[918]:=49.980;
	stepTestFull[919]:=49.980;
	stepTestFull[920]:=49.980;
	stepTestFull[921]:=49.980;
	stepTestFull[922]:=49.980;
	stepTestFull[923]:=49.980;
	stepTestFull[924]:=49.980;
	stepTestFull[925]:=49.980;
	stepTestFull[926]:=49.980;
	stepTestFull[927]:=49.980;
	stepTestFull[928]:=49.980;
	stepTestFull[929]:=49.980;
	stepTestFull[930]:=50.000;
	stepTestFull[931]:=50.000;
	stepTestFull[932]:=50.000;
	stepTestFull[933]:=50.000;
	stepTestFull[934]:=50.000;
	stepTestFull[935]:=50.000;
	stepTestFull[936]:=50.000;
	stepTestFull[937]:=50.000;
	stepTestFull[938]:=50.000;
	stepTestFull[939]:=50.000;
	stepTestFull[940]:=50.000;
	stepTestFull[941]:=50.000;
	stepTestFull[942]:=50.000;
	stepTestFull[943]:=50.000;
	stepTestFull[944]:=50.000;
	stepTestFull[945]:=50.000;
	stepTestFull[946]:=50.000;
	stepTestFull[947]:=50.000;
	stepTestFull[948]:=50.000;
	stepTestFull[949]:=50.000;
	stepTestFull[950]:=50.000;
	stepTestFull[951]:=50.000;
	stepTestFull[952]:=50.000;
	stepTestFull[953]:=50.000;
	stepTestFull[954]:=50.000;
	stepTestFull[955]:=50.000;
	stepTestFull[956]:=50.000;
	stepTestFull[957]:=50.000;
	stepTestFull[958]:=50.000;
	stepTestFull[959]:=50.000;
	stepTestFull[960]:=50.000;
	stepTestFull[961]:=50.000;
	stepTestFull[962]:=50.000;
	stepTestFull[963]:=50.000;
	stepTestFull[964]:=50.000;
	stepTestFull[965]:=50.000;
	stepTestFull[966]:=50.000;
	stepTestFull[967]:=50.000;
	stepTestFull[968]:=50.000;
	stepTestFull[969]:=50.000;
	stepTestFull[970]:=50.000;
	stepTestFull[971]:=50.000;
	stepTestFull[972]:=50.000;
	stepTestFull[973]:=50.000;
	stepTestFull[974]:=50.000;
	stepTestFull[975]:=50.000;
	stepTestFull[976]:=50.000;
	stepTestFull[977]:=50.000;
	stepTestFull[978]:=50.000;
	stepTestFull[979]:=50.000;
	stepTestFull[980]:=50.000;
	stepTestFull[981]:=50.000;
	stepTestFull[982]:=50.000;
	stepTestFull[983]:=50.000;
	stepTestFull[984]:=50.000;
	stepTestFull[985]:=50.000;
	stepTestFull[986]:=50.000;
	stepTestFull[987]:=50.000;
	stepTestFull[988]:=50.000;
	stepTestFull[989]:=50.000;
	stepTestFull[990]:=50.100;
	stepTestFull[991]:=50.100;
	stepTestFull[992]:=50.100;
	stepTestFull[993]:=50.100;
	stepTestFull[994]:=50.100;
	stepTestFull[995]:=50.100;
	stepTestFull[996]:=50.100;
	stepTestFull[997]:=50.100;
	stepTestFull[998]:=50.100;
	stepTestFull[999]:=50.100;
	stepTestFull[1000]:=50.100;
	stepTestFull[1001]:=50.100;
	stepTestFull[1002]:=50.100;
	stepTestFull[1003]:=50.100;
	stepTestFull[1004]:=50.100;
	stepTestFull[1005]:=50.100;
	stepTestFull[1006]:=50.100;
	stepTestFull[1007]:=50.100;
	stepTestFull[1008]:=50.100;
	stepTestFull[1009]:=50.100;
	stepTestFull[1010]:=50.100;
	stepTestFull[1011]:=50.100;
	stepTestFull[1012]:=50.100;
	stepTestFull[1013]:=50.100;
	stepTestFull[1014]:=50.100;
	stepTestFull[1015]:=50.100;
	stepTestFull[1016]:=50.100;
	stepTestFull[1017]:=50.100;
	stepTestFull[1018]:=50.100;
	stepTestFull[1019]:=50.100;
	stepTestFull[1020]:=50.100;
	stepTestFull[1021]:=50.100;
	stepTestFull[1022]:=50.100;
	stepTestFull[1023]:=50.100;
	stepTestFull[1024]:=50.100;
	stepTestFull[1025]:=50.100;
	stepTestFull[1026]:=50.100;
	stepTestFull[1027]:=50.100;
	stepTestFull[1028]:=50.100;
	stepTestFull[1029]:=50.100;
	stepTestFull[1030]:=50.100;
	stepTestFull[1031]:=50.100;
	stepTestFull[1032]:=50.100;
	stepTestFull[1033]:=50.100;
	stepTestFull[1034]:=50.100;
	stepTestFull[1035]:=50.100;
	stepTestFull[1036]:=50.100;
	stepTestFull[1037]:=50.100;
	stepTestFull[1038]:=50.100;
	stepTestFull[1039]:=50.100;
	stepTestFull[1040]:=50.100;
	stepTestFull[1041]:=50.100;
	stepTestFull[1042]:=50.100;
	stepTestFull[1043]:=50.100;
	stepTestFull[1044]:=50.100;
	stepTestFull[1045]:=50.100;
	stepTestFull[1046]:=50.100;
	stepTestFull[1047]:=50.100;
	stepTestFull[1048]:=50.100;
	stepTestFull[1049]:=50.100;
	stepTestFull[1050]:=50.100;
	stepTestFull[1051]:=50.100;
	stepTestFull[1052]:=50.100;
	stepTestFull[1053]:=50.100;
	stepTestFull[1054]:=50.100;
	stepTestFull[1055]:=50.100;
	stepTestFull[1056]:=50.100;
	stepTestFull[1057]:=50.100;
	stepTestFull[1058]:=50.100;
	stepTestFull[1059]:=50.100;
	stepTestFull[1060]:=50.100;
	stepTestFull[1061]:=50.100;
	stepTestFull[1062]:=50.100;
	stepTestFull[1063]:=50.100;
	stepTestFull[1064]:=50.100;
	stepTestFull[1065]:=50.100;
	stepTestFull[1066]:=50.100;
	stepTestFull[1067]:=50.100;
	stepTestFull[1068]:=50.100;
	stepTestFull[1069]:=50.100;
	stepTestFull[1070]:=50.100;
	stepTestFull[1071]:=50.100;
	stepTestFull[1072]:=50.100;
	stepTestFull[1073]:=50.100;
	stepTestFull[1074]:=50.100;
	stepTestFull[1075]:=50.100;
	stepTestFull[1076]:=50.100;
	stepTestFull[1077]:=50.100;
	stepTestFull[1078]:=50.100;
	stepTestFull[1079]:=50.100;
	stepTestFull[1080]:=50.100;
	stepTestFull[1081]:=50.100;
	stepTestFull[1082]:=50.100;
	stepTestFull[1083]:=50.100;
	stepTestFull[1084]:=50.100;
	stepTestFull[1085]:=50.100;
	stepTestFull[1086]:=50.100;
	stepTestFull[1087]:=50.100;
	stepTestFull[1088]:=50.100;
	stepTestFull[1089]:=50.100;
	stepTestFull[1090]:=50.100;
	stepTestFull[1091]:=50.100;
	stepTestFull[1092]:=50.100;
	stepTestFull[1093]:=50.100;
	stepTestFull[1094]:=50.100;
	stepTestFull[1095]:=50.100;
	stepTestFull[1096]:=50.100;
	stepTestFull[1097]:=50.100;
	stepTestFull[1098]:=50.100;
	stepTestFull[1099]:=50.100;
	stepTestFull[1100]:=50.100;
	stepTestFull[1101]:=50.100;
	stepTestFull[1102]:=50.100;
	stepTestFull[1103]:=50.100;
	stepTestFull[1104]:=50.100;
	stepTestFull[1105]:=50.100;
	stepTestFull[1106]:=50.100;
	stepTestFull[1107]:=50.100;
	stepTestFull[1108]:=50.100;
	stepTestFull[1109]:=50.100;
	stepTestFull[1110]:=50.100;
	stepTestFull[1111]:=50.100;
	stepTestFull[1112]:=50.100;
	stepTestFull[1113]:=50.100;
	stepTestFull[1114]:=50.100;
	stepTestFull[1115]:=50.100;
	stepTestFull[1116]:=50.100;
	stepTestFull[1117]:=50.100;
	stepTestFull[1118]:=50.100;
	stepTestFull[1119]:=50.100;
	stepTestFull[1120]:=50.100;
	stepTestFull[1121]:=50.100;
	stepTestFull[1122]:=50.100;
	stepTestFull[1123]:=50.100;
	stepTestFull[1124]:=50.100;
	stepTestFull[1125]:=50.100;
	stepTestFull[1126]:=50.100;
	stepTestFull[1127]:=50.100;
	stepTestFull[1128]:=50.100;
	stepTestFull[1129]:=50.100;
	stepTestFull[1130]:=50.100;
	stepTestFull[1131]:=50.100;
	stepTestFull[1132]:=50.100;
	stepTestFull[1133]:=50.100;
	stepTestFull[1134]:=50.100;
	stepTestFull[1135]:=50.100;
	stepTestFull[1136]:=50.100;
	stepTestFull[1137]:=50.100;
	stepTestFull[1138]:=50.100;
	stepTestFull[1139]:=50.100;
	stepTestFull[1140]:=50.100;
	stepTestFull[1141]:=50.100;
	stepTestFull[1142]:=50.100;
	stepTestFull[1143]:=50.100;
	stepTestFull[1144]:=50.100;
	stepTestFull[1145]:=50.100;
	stepTestFull[1146]:=50.100;
	stepTestFull[1147]:=50.100;
	stepTestFull[1148]:=50.100;
	stepTestFull[1149]:=50.100;
	stepTestFull[1150]:=50.100;
	stepTestFull[1151]:=50.100;
	stepTestFull[1152]:=50.100;
	stepTestFull[1153]:=50.100;
	stepTestFull[1154]:=50.100;
	stepTestFull[1155]:=50.100;
	stepTestFull[1156]:=50.100;
	stepTestFull[1157]:=50.100;
	stepTestFull[1158]:=50.100;
	stepTestFull[1159]:=50.100;
	stepTestFull[1160]:=50.100;
	stepTestFull[1161]:=50.100;
	stepTestFull[1162]:=50.100;
	stepTestFull[1163]:=50.100;
	stepTestFull[1164]:=50.100;
	stepTestFull[1165]:=50.100;
	stepTestFull[1166]:=50.100;
	stepTestFull[1167]:=50.100;
	stepTestFull[1168]:=50.100;
	stepTestFull[1169]:=50.100;
	stepTestFull[1170]:=50.000;
	stepTestFull[1171]:=50.000;
	stepTestFull[1172]:=50.000;
	stepTestFull[1173]:=50.000;
	stepTestFull[1174]:=50.000;
	stepTestFull[1175]:=50.000;
	stepTestFull[1176]:=50.000;
	stepTestFull[1177]:=50.000;
	stepTestFull[1178]:=50.000;
	stepTestFull[1179]:=50.000;
	stepTestFull[1180]:=50.000;
	stepTestFull[1181]:=50.000;
	stepTestFull[1182]:=50.000;
	stepTestFull[1183]:=50.000;
	stepTestFull[1184]:=50.000;
	stepTestFull[1185]:=50.000;
	stepTestFull[1186]:=50.000;
	stepTestFull[1187]:=50.000;
	stepTestFull[1188]:=50.000;
	stepTestFull[1189]:=50.000;
	stepTestFull[1190]:=50.000;
	stepTestFull[1191]:=50.000;
	stepTestFull[1192]:=50.000;
	stepTestFull[1193]:=50.000;
	stepTestFull[1194]:=50.000;
	stepTestFull[1195]:=50.000;
	stepTestFull[1196]:=50.000;
	stepTestFull[1197]:=50.000;
	stepTestFull[1198]:=50.000;
	stepTestFull[1199]:=50.000;
	stepTestFull[1200]:=50.000;
	stepTestFull[1201]:=50.000;
	stepTestFull[1202]:=50.000;
	stepTestFull[1203]:=50.000;
	stepTestFull[1204]:=50.000;
	stepTestFull[1205]:=50.000;
	stepTestFull[1206]:=50.000;
	stepTestFull[1207]:=50.000;
	stepTestFull[1208]:=50.000;
	stepTestFull[1209]:=50.000;
	stepTestFull[1210]:=50.000;
	stepTestFull[1211]:=50.000;
	stepTestFull[1212]:=50.000;
	stepTestFull[1213]:=50.000;
	stepTestFull[1214]:=50.000;
	stepTestFull[1215]:=50.000;
	stepTestFull[1216]:=50.000;
	stepTestFull[1217]:=50.000;
	stepTestFull[1218]:=50.000;
	stepTestFull[1219]:=50.000;
	stepTestFull[1220]:=50.000;
	stepTestFull[1221]:=50.000;
	stepTestFull[1222]:=50.000;
	stepTestFull[1223]:=50.000;
	stepTestFull[1224]:=50.000;
	stepTestFull[1225]:=50.000;
	stepTestFull[1226]:=50.000;
	stepTestFull[1227]:=50.000;
	stepTestFull[1228]:=50.000;
	stepTestFull[1229]:=50.000;
	stepTestFull[1230]:=49.900;
	stepTestFull[1231]:=49.900;
	stepTestFull[1232]:=49.900;
	stepTestFull[1233]:=49.900;
	stepTestFull[1234]:=49.900;
	stepTestFull[1235]:=49.900;
	stepTestFull[1236]:=49.900;
	stepTestFull[1237]:=49.900;
	stepTestFull[1238]:=49.900;
	stepTestFull[1239]:=49.900;
	stepTestFull[1240]:=49.900;
	stepTestFull[1241]:=49.900;
	stepTestFull[1242]:=49.900;
	stepTestFull[1243]:=49.900;
	stepTestFull[1244]:=49.900;
	stepTestFull[1245]:=49.900;
	stepTestFull[1246]:=49.900;
	stepTestFull[1247]:=49.900;
	stepTestFull[1248]:=49.900;
	stepTestFull[1249]:=49.900;
	stepTestFull[1250]:=49.900;
	stepTestFull[1251]:=49.900;
	stepTestFull[1252]:=49.900;
	stepTestFull[1253]:=49.900;
	stepTestFull[1254]:=49.900;
	stepTestFull[1255]:=49.900;
	stepTestFull[1256]:=49.900;
	stepTestFull[1257]:=49.900;
	stepTestFull[1258]:=49.900;
	stepTestFull[1259]:=49.900;
	stepTestFull[1260]:=49.900;
	stepTestFull[1261]:=49.900;
	stepTestFull[1262]:=49.900;
	stepTestFull[1263]:=49.900;
	stepTestFull[1264]:=49.900;
	stepTestFull[1265]:=49.900;
	stepTestFull[1266]:=49.900;
	stepTestFull[1267]:=49.900;
	stepTestFull[1268]:=49.900;
	stepTestFull[1269]:=49.900;
	stepTestFull[1270]:=49.900;
	stepTestFull[1271]:=49.900;
	stepTestFull[1272]:=49.900;
	stepTestFull[1273]:=49.900;
	stepTestFull[1274]:=49.900;
	stepTestFull[1275]:=49.900;
	stepTestFull[1276]:=49.900;
	stepTestFull[1277]:=49.900;
	stepTestFull[1278]:=49.900;
	stepTestFull[1279]:=49.900;
	stepTestFull[1280]:=49.900;
	stepTestFull[1281]:=49.900;
	stepTestFull[1282]:=49.900;
	stepTestFull[1283]:=49.900;
	stepTestFull[1284]:=49.900;
	stepTestFull[1285]:=49.900;
	stepTestFull[1286]:=49.900;
	stepTestFull[1287]:=49.900;
	stepTestFull[1288]:=49.900;
	stepTestFull[1289]:=49.900;
	stepTestFull[1290]:=49.900;
	stepTestFull[1291]:=49.900;
	stepTestFull[1292]:=49.900;
	stepTestFull[1293]:=49.900;
	stepTestFull[1294]:=49.900;
	stepTestFull[1295]:=49.900;
	stepTestFull[1296]:=49.900;
	stepTestFull[1297]:=49.900;
	stepTestFull[1298]:=49.900;
	stepTestFull[1299]:=49.900;
	stepTestFull[1300]:=49.900;
	stepTestFull[1301]:=49.900;
	stepTestFull[1302]:=49.900;
	stepTestFull[1303]:=49.900;
	stepTestFull[1304]:=49.900;
	stepTestFull[1305]:=49.900;
	stepTestFull[1306]:=49.900;
	stepTestFull[1307]:=49.900;
	stepTestFull[1308]:=49.900;
	stepTestFull[1309]:=49.900;
	stepTestFull[1310]:=49.900;
	stepTestFull[1311]:=49.900;
	stepTestFull[1312]:=49.900;
	stepTestFull[1313]:=49.900;
	stepTestFull[1314]:=49.900;
	stepTestFull[1315]:=49.900;
	stepTestFull[1316]:=49.900;
	stepTestFull[1317]:=49.900;
	stepTestFull[1318]:=49.900;
	stepTestFull[1319]:=49.900;
	stepTestFull[1320]:=49.900;
	stepTestFull[1321]:=49.900;
	stepTestFull[1322]:=49.900;
	stepTestFull[1323]:=49.900;
	stepTestFull[1324]:=49.900;
	stepTestFull[1325]:=49.900;
	stepTestFull[1326]:=49.900;
	stepTestFull[1327]:=49.900;
	stepTestFull[1328]:=49.900;
	stepTestFull[1329]:=49.900;
	stepTestFull[1330]:=49.900;
	stepTestFull[1331]:=49.900;
	stepTestFull[1332]:=49.900;
	stepTestFull[1333]:=49.900;
	stepTestFull[1334]:=49.900;
	stepTestFull[1335]:=49.900;
	stepTestFull[1336]:=49.900;
	stepTestFull[1337]:=49.900;
	stepTestFull[1338]:=49.900;
	stepTestFull[1339]:=49.900;
	stepTestFull[1340]:=49.900;
	stepTestFull[1341]:=49.900;
	stepTestFull[1342]:=49.900;
	stepTestFull[1343]:=49.900;
	stepTestFull[1344]:=49.900;
	stepTestFull[1345]:=49.900;
	stepTestFull[1346]:=49.900;
	stepTestFull[1347]:=49.900;
	stepTestFull[1348]:=49.900;
	stepTestFull[1349]:=49.900;
	stepTestFull[1350]:=49.900;
	stepTestFull[1351]:=49.900;
	stepTestFull[1352]:=49.900;
	stepTestFull[1353]:=49.900;
	stepTestFull[1354]:=49.900;
	stepTestFull[1355]:=49.900;
	stepTestFull[1356]:=49.900;
	stepTestFull[1357]:=49.900;
	stepTestFull[1358]:=49.900;
	stepTestFull[1359]:=49.900;
	stepTestFull[1360]:=49.900;
	stepTestFull[1361]:=49.900;
	stepTestFull[1362]:=49.900;
	stepTestFull[1363]:=49.900;
	stepTestFull[1364]:=49.900;
	stepTestFull[1365]:=49.900;
	stepTestFull[1366]:=49.900;
	stepTestFull[1367]:=49.900;
	stepTestFull[1368]:=49.900;
	stepTestFull[1369]:=49.900;
	stepTestFull[1370]:=49.900;
	stepTestFull[1371]:=49.900;
	stepTestFull[1372]:=49.900;
	stepTestFull[1373]:=49.900;
	stepTestFull[1374]:=49.900;
	stepTestFull[1375]:=49.900;
	stepTestFull[1376]:=49.900;
	stepTestFull[1377]:=49.900;
	stepTestFull[1378]:=49.900;
	stepTestFull[1379]:=49.900;
	stepTestFull[1380]:=49.900;
	stepTestFull[1381]:=49.900;
	stepTestFull[1382]:=49.900;
	stepTestFull[1383]:=49.900;
	stepTestFull[1384]:=49.900;
	stepTestFull[1385]:=49.900;
	stepTestFull[1386]:=49.900;
	stepTestFull[1387]:=49.900;
	stepTestFull[1388]:=49.900;
	stepTestFull[1389]:=49.900;
	stepTestFull[1390]:=49.900;
	stepTestFull[1391]:=49.900;
	stepTestFull[1392]:=49.900;
	stepTestFull[1393]:=49.900;
	stepTestFull[1394]:=49.900;
	stepTestFull[1395]:=49.900;
	stepTestFull[1396]:=49.900;
	stepTestFull[1397]:=49.900;
	stepTestFull[1398]:=49.900;
	stepTestFull[1399]:=49.900;
	stepTestFull[1400]:=49.900;
	stepTestFull[1401]:=49.900;
	stepTestFull[1402]:=49.900;
	stepTestFull[1403]:=49.900;
	stepTestFull[1404]:=49.900;
	stepTestFull[1405]:=49.900;
	stepTestFull[1406]:=49.900;
	stepTestFull[1407]:=49.900;
	stepTestFull[1408]:=49.900;
	stepTestFull[1409]:=49.900;
	stepTestFull[1410]:=50.000;
	stepTestFull[1411]:=50.000;
	stepTestFull[1412]:=50.000;
	stepTestFull[1413]:=50.000;
	stepTestFull[1414]:=50.000;
	stepTestFull[1415]:=50.000;
	stepTestFull[1416]:=50.000;
	stepTestFull[1417]:=50.000;
	stepTestFull[1418]:=50.000;
	stepTestFull[1419]:=50.000;
	stepTestFull[1420]:=50.000;
	stepTestFull[1421]:=50.000;
	stepTestFull[1422]:=50.000;
	stepTestFull[1423]:=50.000;
	stepTestFull[1424]:=50.000;
	stepTestFull[1425]:=50.000;
	stepTestFull[1426]:=50.000;
	stepTestFull[1427]:=50.000;
	stepTestFull[1428]:=50.000;
	stepTestFull[1429]:=50.000;
	stepTestFull[1430]:=50.000;
	stepTestFull[1431]:=50.000;
	stepTestFull[1432]:=50.000;
	stepTestFull[1433]:=50.000;
	stepTestFull[1434]:=50.000;
	stepTestFull[1435]:=50.000;
	stepTestFull[1436]:=50.000;
	stepTestFull[1437]:=50.000;
	stepTestFull[1438]:=50.000;
	stepTestFull[1439]:=50.000;
	stepTestFull[1440]:=50.000;
	stepTestFull[1441]:=50.000;
	stepTestFull[1442]:=50.000;
	stepTestFull[1443]:=50.000;
	stepTestFull[1444]:=50.000;
	stepTestFull[1445]:=50.000;
	stepTestFull[1446]:=50.000;
	stepTestFull[1447]:=50.000;
	stepTestFull[1448]:=50.000;
	stepTestFull[1449]:=50.000;
	stepTestFull[1450]:=50.000;
	stepTestFull[1451]:=50.000;
	stepTestFull[1452]:=50.000;
	stepTestFull[1453]:=50.000;
	stepTestFull[1454]:=50.000;
	stepTestFull[1455]:=50.000;
	stepTestFull[1456]:=50.000;
	stepTestFull[1457]:=50.000;
	stepTestFull[1458]:=50.000;
	stepTestFull[1459]:=50.000;
	stepTestFull[1460]:=50.000;
	stepTestFull[1461]:=50.000;
	stepTestFull[1462]:=50.000;
	stepTestFull[1463]:=50.000;
	stepTestFull[1464]:=50.000;
	stepTestFull[1465]:=50.000;
	stepTestFull[1466]:=50.000;
	stepTestFull[1467]:=50.000;
	stepTestFull[1468]:=50.000;
	stepTestFull[1469]:=50.000;
	stepTestFull[1470]:=50.200;
	stepTestFull[1471]:=50.200;
	stepTestFull[1472]:=50.200;
	stepTestFull[1473]:=50.200;
	stepTestFull[1474]:=50.200;
	stepTestFull[1475]:=50.200;
	stepTestFull[1476]:=50.200;
	stepTestFull[1477]:=50.200;
	stepTestFull[1478]:=50.200;
	stepTestFull[1479]:=50.200;
	stepTestFull[1480]:=50.200;
	stepTestFull[1481]:=50.200;
	stepTestFull[1482]:=50.200;
	stepTestFull[1483]:=50.200;
	stepTestFull[1484]:=50.200;
	stepTestFull[1485]:=50.200;
	stepTestFull[1486]:=50.200;
	stepTestFull[1487]:=50.200;
	stepTestFull[1488]:=50.200;
	stepTestFull[1489]:=50.200;
	stepTestFull[1490]:=50.200;
	stepTestFull[1491]:=50.200;
	stepTestFull[1492]:=50.200;
	stepTestFull[1493]:=50.200;
	stepTestFull[1494]:=50.200;
	stepTestFull[1495]:=50.200;
	stepTestFull[1496]:=50.200;
	stepTestFull[1497]:=50.200;
	stepTestFull[1498]:=50.200;
	stepTestFull[1499]:=50.200;
	stepTestFull[1500]:=50.200;
	stepTestFull[1501]:=50.200;
	stepTestFull[1502]:=50.200;
	stepTestFull[1503]:=50.200;
	stepTestFull[1504]:=50.200;
	stepTestFull[1505]:=50.200;
	stepTestFull[1506]:=50.200;
	stepTestFull[1507]:=50.200;
	stepTestFull[1508]:=50.200;
	stepTestFull[1509]:=50.200;
	stepTestFull[1510]:=50.200;
	stepTestFull[1511]:=50.200;
	stepTestFull[1512]:=50.200;
	stepTestFull[1513]:=50.200;
	stepTestFull[1514]:=50.200;
	stepTestFull[1515]:=50.200;
	stepTestFull[1516]:=50.200;
	stepTestFull[1517]:=50.200;
	stepTestFull[1518]:=50.200;
	stepTestFull[1519]:=50.200;
	stepTestFull[1520]:=50.200;
	stepTestFull[1521]:=50.200;
	stepTestFull[1522]:=50.200;
	stepTestFull[1523]:=50.200;
	stepTestFull[1524]:=50.200;
	stepTestFull[1525]:=50.200;
	stepTestFull[1526]:=50.200;
	stepTestFull[1527]:=50.200;
	stepTestFull[1528]:=50.200;
	stepTestFull[1529]:=50.200;
	stepTestFull[1530]:=50.200;
	stepTestFull[1531]:=50.200;
	stepTestFull[1532]:=50.200;
	stepTestFull[1533]:=50.200;
	stepTestFull[1534]:=50.200;
	stepTestFull[1535]:=50.200;
	stepTestFull[1536]:=50.200;
	stepTestFull[1537]:=50.200;
	stepTestFull[1538]:=50.200;
	stepTestFull[1539]:=50.200;
	stepTestFull[1540]:=50.200;
	stepTestFull[1541]:=50.200;
	stepTestFull[1542]:=50.200;
	stepTestFull[1543]:=50.200;
	stepTestFull[1544]:=50.200;
	stepTestFull[1545]:=50.200;
	stepTestFull[1546]:=50.200;
	stepTestFull[1547]:=50.200;
	stepTestFull[1548]:=50.200;
	stepTestFull[1549]:=50.200;
	stepTestFull[1550]:=50.200;
	stepTestFull[1551]:=50.200;
	stepTestFull[1552]:=50.200;
	stepTestFull[1553]:=50.200;
	stepTestFull[1554]:=50.200;
	stepTestFull[1555]:=50.200;
	stepTestFull[1556]:=50.200;
	stepTestFull[1557]:=50.200;
	stepTestFull[1558]:=50.200;
	stepTestFull[1559]:=50.200;
	stepTestFull[1560]:=50.200;
	stepTestFull[1561]:=50.200;
	stepTestFull[1562]:=50.200;
	stepTestFull[1563]:=50.200;
	stepTestFull[1564]:=50.200;
	stepTestFull[1565]:=50.200;
	stepTestFull[1566]:=50.200;
	stepTestFull[1567]:=50.200;
	stepTestFull[1568]:=50.200;
	stepTestFull[1569]:=50.200;
	stepTestFull[1570]:=50.200;
	stepTestFull[1571]:=50.200;
	stepTestFull[1572]:=50.200;
	stepTestFull[1573]:=50.200;
	stepTestFull[1574]:=50.200;
	stepTestFull[1575]:=50.200;
	stepTestFull[1576]:=50.200;
	stepTestFull[1577]:=50.200;
	stepTestFull[1578]:=50.200;
	stepTestFull[1579]:=50.200;
	stepTestFull[1580]:=50.200;
	stepTestFull[1581]:=50.200;
	stepTestFull[1582]:=50.200;
	stepTestFull[1583]:=50.200;
	stepTestFull[1584]:=50.200;
	stepTestFull[1585]:=50.200;
	stepTestFull[1586]:=50.200;
	stepTestFull[1587]:=50.200;
	stepTestFull[1588]:=50.200;
	stepTestFull[1589]:=50.200;
	stepTestFull[1590]:=50.200;
	stepTestFull[1591]:=50.200;
	stepTestFull[1592]:=50.200;
	stepTestFull[1593]:=50.200;
	stepTestFull[1594]:=50.200;
	stepTestFull[1595]:=50.200;
	stepTestFull[1596]:=50.200;
	stepTestFull[1597]:=50.200;
	stepTestFull[1598]:=50.200;
	stepTestFull[1599]:=50.200;
	stepTestFull[1600]:=50.200;
	stepTestFull[1601]:=50.200;
	stepTestFull[1602]:=50.200;
	stepTestFull[1603]:=50.200;
	stepTestFull[1604]:=50.200;
	stepTestFull[1605]:=50.200;
	stepTestFull[1606]:=50.200;
	stepTestFull[1607]:=50.200;
	stepTestFull[1608]:=50.200;
	stepTestFull[1609]:=50.200;
	stepTestFull[1610]:=50.200;
	stepTestFull[1611]:=50.200;
	stepTestFull[1612]:=50.200;
	stepTestFull[1613]:=50.200;
	stepTestFull[1614]:=50.200;
	stepTestFull[1615]:=50.200;
	stepTestFull[1616]:=50.200;
	stepTestFull[1617]:=50.200;
	stepTestFull[1618]:=50.200;
	stepTestFull[1619]:=50.200;
	stepTestFull[1620]:=50.200;
	stepTestFull[1621]:=50.200;
	stepTestFull[1622]:=50.200;
	stepTestFull[1623]:=50.200;
	stepTestFull[1624]:=50.200;
	stepTestFull[1625]:=50.200;
	stepTestFull[1626]:=50.200;
	stepTestFull[1627]:=50.200;
	stepTestFull[1628]:=50.200;
	stepTestFull[1629]:=50.200;
	stepTestFull[1630]:=50.200;
	stepTestFull[1631]:=50.200;
	stepTestFull[1632]:=50.200;
	stepTestFull[1633]:=50.200;
	stepTestFull[1634]:=50.200;
	stepTestFull[1635]:=50.200;
	stepTestFull[1636]:=50.200;
	stepTestFull[1637]:=50.200;
	stepTestFull[1638]:=50.200;
	stepTestFull[1639]:=50.200;
	stepTestFull[1640]:=50.200;
	stepTestFull[1641]:=50.200;
	stepTestFull[1642]:=50.200;
	stepTestFull[1643]:=50.200;
	stepTestFull[1644]:=50.200;
	stepTestFull[1645]:=50.200;
	stepTestFull[1646]:=50.200;
	stepTestFull[1647]:=50.200;
	stepTestFull[1648]:=50.200;
	stepTestFull[1649]:=50.200;
	stepTestFull[1650]:=50.000;
	stepTestFull[1651]:=50.000;
	stepTestFull[1652]:=50.000;
	stepTestFull[1653]:=50.000;
	stepTestFull[1654]:=50.000;
	stepTestFull[1655]:=50.000;
	stepTestFull[1656]:=50.000;
	stepTestFull[1657]:=50.000;
	stepTestFull[1658]:=50.000;
	stepTestFull[1659]:=50.000;
	stepTestFull[1660]:=50.000;
	stepTestFull[1661]:=50.000;
	stepTestFull[1662]:=50.000;
	stepTestFull[1663]:=50.000;
	stepTestFull[1664]:=50.000;
	stepTestFull[1665]:=50.000;
	stepTestFull[1666]:=50.000;
	stepTestFull[1667]:=50.000;
	stepTestFull[1668]:=50.000;
	stepTestFull[1669]:=50.000;
	stepTestFull[1670]:=50.000;
	stepTestFull[1671]:=50.000;
	stepTestFull[1672]:=50.000;
	stepTestFull[1673]:=50.000;
	stepTestFull[1674]:=50.000;
	stepTestFull[1675]:=50.000;
	stepTestFull[1676]:=50.000;
	stepTestFull[1677]:=50.000;
	stepTestFull[1678]:=50.000;
	stepTestFull[1679]:=50.000;
	stepTestFull[1680]:=50.000;
	stepTestFull[1681]:=50.000;
	stepTestFull[1682]:=50.000;
	stepTestFull[1683]:=50.000;
	stepTestFull[1684]:=50.000;
	stepTestFull[1685]:=50.000;
	stepTestFull[1686]:=50.000;
	stepTestFull[1687]:=50.000;
	stepTestFull[1688]:=50.000;
	stepTestFull[1689]:=50.000;
	stepTestFull[1690]:=50.000;
	stepTestFull[1691]:=50.000;
	stepTestFull[1692]:=50.000;
	stepTestFull[1693]:=50.000;
	stepTestFull[1694]:=50.000;
	stepTestFull[1695]:=50.000;
	stepTestFull[1696]:=50.000;
	stepTestFull[1697]:=50.000;
	stepTestFull[1698]:=50.000;
	stepTestFull[1699]:=50.000;
	stepTestFull[1700]:=50.000;
	stepTestFull[1701]:=50.000;
	stepTestFull[1702]:=50.000;
	stepTestFull[1703]:=50.000;
	stepTestFull[1704]:=50.000;
	stepTestFull[1705]:=50.000;
	stepTestFull[1706]:=50.000;
	stepTestFull[1707]:=50.000;
	stepTestFull[1708]:=50.000;
	stepTestFull[1709]:=50.000;
	stepTestFull[1710]:=49.800;
	stepTestFull[1711]:=49.800;
	stepTestFull[1712]:=49.800;
	stepTestFull[1713]:=49.800;
	stepTestFull[1714]:=49.800;
	stepTestFull[1715]:=49.800;
	stepTestFull[1716]:=49.800;
	stepTestFull[1717]:=49.800;
	stepTestFull[1718]:=49.800;
	stepTestFull[1719]:=49.800;
	stepTestFull[1720]:=49.800;
	stepTestFull[1721]:=49.800;
	stepTestFull[1722]:=49.800;
	stepTestFull[1723]:=49.800;
	stepTestFull[1724]:=49.800;
	stepTestFull[1725]:=49.800;
	stepTestFull[1726]:=49.800;
	stepTestFull[1727]:=49.800;
	stepTestFull[1728]:=49.800;
	stepTestFull[1729]:=49.800;
	stepTestFull[1730]:=49.800;
	stepTestFull[1731]:=49.800;
	stepTestFull[1732]:=49.800;
	stepTestFull[1733]:=49.800;
	stepTestFull[1734]:=49.800;
	stepTestFull[1735]:=49.800;
	stepTestFull[1736]:=49.800;
	stepTestFull[1737]:=49.800;
	stepTestFull[1738]:=49.800;
	stepTestFull[1739]:=49.800;
	stepTestFull[1740]:=49.800;
	stepTestFull[1741]:=49.800;
	stepTestFull[1742]:=49.800;
	stepTestFull[1743]:=49.800;
	stepTestFull[1744]:=49.800;
	stepTestFull[1745]:=49.800;
	stepTestFull[1746]:=49.800;
	stepTestFull[1747]:=49.800;
	stepTestFull[1748]:=49.800;
	stepTestFull[1749]:=49.800;
	stepTestFull[1750]:=49.800;
	stepTestFull[1751]:=49.800;
	stepTestFull[1752]:=49.800;
	stepTestFull[1753]:=49.800;
	stepTestFull[1754]:=49.800;
	stepTestFull[1755]:=49.800;
	stepTestFull[1756]:=49.800;
	stepTestFull[1757]:=49.800;
	stepTestFull[1758]:=49.800;
	stepTestFull[1759]:=49.800;
	stepTestFull[1760]:=49.800;
	stepTestFull[1761]:=49.800;
	stepTestFull[1762]:=49.800;
	stepTestFull[1763]:=49.800;
	stepTestFull[1764]:=49.800;
	stepTestFull[1765]:=49.800;
	stepTestFull[1766]:=49.800;
	stepTestFull[1767]:=49.800;
	stepTestFull[1768]:=49.800;
	stepTestFull[1769]:=49.800;
	stepTestFull[1770]:=49.800;
	stepTestFull[1771]:=49.800;
	stepTestFull[1772]:=49.800;
	stepTestFull[1773]:=49.800;
	stepTestFull[1774]:=49.800;
	stepTestFull[1775]:=49.800;
	stepTestFull[1776]:=49.800;
	stepTestFull[1777]:=49.800;
	stepTestFull[1778]:=49.800;
	stepTestFull[1779]:=49.800;
	stepTestFull[1780]:=49.800;
	stepTestFull[1781]:=49.800;
	stepTestFull[1782]:=49.800;
	stepTestFull[1783]:=49.800;
	stepTestFull[1784]:=49.800;
	stepTestFull[1785]:=49.800;
	stepTestFull[1786]:=49.800;
	stepTestFull[1787]:=49.800;
	stepTestFull[1788]:=49.800;
	stepTestFull[1789]:=49.800;
	stepTestFull[1790]:=49.800;
	stepTestFull[1791]:=49.800;
	stepTestFull[1792]:=49.800;
	stepTestFull[1793]:=49.800;
	stepTestFull[1794]:=49.800;
	stepTestFull[1795]:=49.800;
	stepTestFull[1796]:=49.800;
	stepTestFull[1797]:=49.800;
	stepTestFull[1798]:=49.800;
	stepTestFull[1799]:=49.800;
	stepTestFull[1800]:=49.800;
	stepTestFull[1801]:=49.800;
	stepTestFull[1802]:=49.800;
	stepTestFull[1803]:=49.800;
	stepTestFull[1804]:=49.800;
	stepTestFull[1805]:=49.800;
	stepTestFull[1806]:=49.800;
	stepTestFull[1807]:=49.800;
	stepTestFull[1808]:=49.800;
	stepTestFull[1809]:=49.800;
	stepTestFull[1810]:=49.800;
	stepTestFull[1811]:=49.800;
	stepTestFull[1812]:=49.800;
	stepTestFull[1813]:=49.800;
	stepTestFull[1814]:=49.800;
	stepTestFull[1815]:=49.800;
	stepTestFull[1816]:=49.800;
	stepTestFull[1817]:=49.800;
	stepTestFull[1818]:=49.800;
	stepTestFull[1819]:=49.800;
	stepTestFull[1820]:=49.800;
	stepTestFull[1821]:=49.800;
	stepTestFull[1822]:=49.800;
	stepTestFull[1823]:=49.800;
	stepTestFull[1824]:=49.800;
	stepTestFull[1825]:=49.800;
	stepTestFull[1826]:=49.800;
	stepTestFull[1827]:=49.800;
	stepTestFull[1828]:=49.800;
	stepTestFull[1829]:=49.800;
	stepTestFull[1830]:=49.800;
	stepTestFull[1831]:=49.800;
	stepTestFull[1832]:=49.800;
	stepTestFull[1833]:=49.800;
	stepTestFull[1834]:=49.800;
	stepTestFull[1835]:=49.800;
	stepTestFull[1836]:=49.800;
	stepTestFull[1837]:=49.800;
	stepTestFull[1838]:=49.800;
	stepTestFull[1839]:=49.800;
	stepTestFull[1840]:=49.800;
	stepTestFull[1841]:=49.800;
	stepTestFull[1842]:=49.800;
	stepTestFull[1843]:=49.800;
	stepTestFull[1844]:=49.800;
	stepTestFull[1845]:=49.800;
	stepTestFull[1846]:=49.800;
	stepTestFull[1847]:=49.800;
	stepTestFull[1848]:=49.800;
	stepTestFull[1849]:=49.800;
	stepTestFull[1850]:=49.800;
	stepTestFull[1851]:=49.800;
	stepTestFull[1852]:=49.800;
	stepTestFull[1853]:=49.800;
	stepTestFull[1854]:=49.800;
	stepTestFull[1855]:=49.800;
	stepTestFull[1856]:=49.800;
	stepTestFull[1857]:=49.800;
	stepTestFull[1858]:=49.800;
	stepTestFull[1859]:=49.800;
	stepTestFull[1860]:=49.800;
	stepTestFull[1861]:=49.800;
	stepTestFull[1862]:=49.800;
	stepTestFull[1863]:=49.800;
	stepTestFull[1864]:=49.800;
	stepTestFull[1865]:=49.800;
	stepTestFull[1866]:=49.800;
	stepTestFull[1867]:=49.800;
	stepTestFull[1868]:=49.800;
	stepTestFull[1869]:=49.800;
	stepTestFull[1870]:=49.800;
	stepTestFull[1871]:=49.800;
	stepTestFull[1872]:=49.800;
	stepTestFull[1873]:=49.800;
	stepTestFull[1874]:=49.800;
	stepTestFull[1875]:=49.800;
	stepTestFull[1876]:=49.800;
	stepTestFull[1877]:=49.800;
	stepTestFull[1878]:=49.800;
	stepTestFull[1879]:=49.800;
	stepTestFull[1880]:=49.800;
	stepTestFull[1881]:=49.800;
	stepTestFull[1882]:=49.800;
	stepTestFull[1883]:=49.800;
	stepTestFull[1884]:=49.800;
	stepTestFull[1885]:=49.800;
	stepTestFull[1886]:=49.800;
	stepTestFull[1887]:=49.800;
	stepTestFull[1888]:=49.800;
	stepTestFull[1889]:=49.800;
	stepTestFull[1890]:=50.000;
	stepTestFull[1891]:=50.000;
	stepTestFull[1892]:=50.000;
	stepTestFull[1893]:=50.000;
	stepTestFull[1894]:=50.000;
	stepTestFull[1895]:=50.000;
	stepTestFull[1896]:=50.000;
	stepTestFull[1897]:=50.000;
	stepTestFull[1898]:=50.000;
	stepTestFull[1899]:=50.000;
	stepTestFull[1900]:=50.000;
	stepTestFull[1901]:=50.000;
	stepTestFull[1902]:=50.000;
	stepTestFull[1903]:=50.000;
	stepTestFull[1904]:=50.000;
	stepTestFull[1905]:=50.000;
	stepTestFull[1906]:=50.000;
	stepTestFull[1907]:=50.000;
	stepTestFull[1908]:=50.000;
	stepTestFull[1909]:=50.000;
	stepTestFull[1910]:=50.000;
	stepTestFull[1911]:=50.000;
	stepTestFull[1912]:=50.000;
	stepTestFull[1913]:=50.000;
	stepTestFull[1914]:=50.000;
	stepTestFull[1915]:=50.000;
	stepTestFull[1916]:=50.000;
	stepTestFull[1917]:=50.000;
	stepTestFull[1918]:=50.000;
	stepTestFull[1919]:=50.000;
	stepTestFull[1920]:=50.000;
	stepTestFull[1921]:=50.000;
	stepTestFull[1922]:=50.000;
	stepTestFull[1923]:=50.000;
	stepTestFull[1924]:=50.000;
	stepTestFull[1925]:=50.000;
	stepTestFull[1926]:=50.000;
	stepTestFull[1927]:=50.000;
	stepTestFull[1928]:=50.000;
	stepTestFull[1929]:=50.000;
	stepTestFull[1930]:=50.000;
	stepTestFull[1931]:=50.000;
	stepTestFull[1932]:=50.000;
	stepTestFull[1933]:=50.000;
	stepTestFull[1934]:=50.000;
	stepTestFull[1935]:=50.000;
	stepTestFull[1936]:=50.000;
	stepTestFull[1937]:=50.000;
	stepTestFull[1938]:=50.000;
	stepTestFull[1939]:=50.000;
	stepTestFull[1940]:=50.000;
	stepTestFull[1941]:=50.000;
	stepTestFull[1942]:=50.000;
	stepTestFull[1943]:=50.000;
	stepTestFull[1944]:=50.000;
	stepTestFull[1945]:=50.000;
	stepTestFull[1946]:=50.000;
	stepTestFull[1947]:=50.000;
	stepTestFull[1948]:=50.000;
	stepTestFull[1949]:=50.000;
	stepTestFull[1950]:=50.300;
	stepTestFull[1951]:=50.300;
	stepTestFull[1952]:=50.300;
	stepTestFull[1953]:=50.300;
	stepTestFull[1954]:=50.300;
	stepTestFull[1955]:=50.300;
	stepTestFull[1956]:=50.300;
	stepTestFull[1957]:=50.300;
	stepTestFull[1958]:=50.300;
	stepTestFull[1959]:=50.300;
	stepTestFull[1960]:=50.300;
	stepTestFull[1961]:=50.300;
	stepTestFull[1962]:=50.300;
	stepTestFull[1963]:=50.300;
	stepTestFull[1964]:=50.300;
	stepTestFull[1965]:=50.300;
	stepTestFull[1966]:=50.300;
	stepTestFull[1967]:=50.300;
	stepTestFull[1968]:=50.300;
	stepTestFull[1969]:=50.300;
	stepTestFull[1970]:=50.300;
	stepTestFull[1971]:=50.300;
	stepTestFull[1972]:=50.300;
	stepTestFull[1973]:=50.300;
	stepTestFull[1974]:=50.300;
	stepTestFull[1975]:=50.300;
	stepTestFull[1976]:=50.300;
	stepTestFull[1977]:=50.300;
	stepTestFull[1978]:=50.300;
	stepTestFull[1979]:=50.300;
	stepTestFull[1980]:=50.300;
	stepTestFull[1981]:=50.300;
	stepTestFull[1982]:=50.300;
	stepTestFull[1983]:=50.300;
	stepTestFull[1984]:=50.300;
	stepTestFull[1985]:=50.300;
	stepTestFull[1986]:=50.300;
	stepTestFull[1987]:=50.300;
	stepTestFull[1988]:=50.300;
	stepTestFull[1989]:=50.300;
	stepTestFull[1990]:=50.300;
	stepTestFull[1991]:=50.300;
	stepTestFull[1992]:=50.300;
	stepTestFull[1993]:=50.300;
	stepTestFull[1994]:=50.300;
	stepTestFull[1995]:=50.300;
	stepTestFull[1996]:=50.300;
	stepTestFull[1997]:=50.300;
	stepTestFull[1998]:=50.300;
	stepTestFull[1999]:=50.300;
	stepTestFull[2000]:=50.300;
	stepTestFull[2001]:=50.300;
	stepTestFull[2002]:=50.300;
	stepTestFull[2003]:=50.300;
	stepTestFull[2004]:=50.300;
	stepTestFull[2005]:=50.300;
	stepTestFull[2006]:=50.300;
	stepTestFull[2007]:=50.300;
	stepTestFull[2008]:=50.300;
	stepTestFull[2009]:=50.300;
	stepTestFull[2010]:=50.300;
	stepTestFull[2011]:=50.300;
	stepTestFull[2012]:=50.300;
	stepTestFull[2013]:=50.300;
	stepTestFull[2014]:=50.300;
	stepTestFull[2015]:=50.300;
	stepTestFull[2016]:=50.300;
	stepTestFull[2017]:=50.300;
	stepTestFull[2018]:=50.300;
	stepTestFull[2019]:=50.300;
	stepTestFull[2020]:=50.300;
	stepTestFull[2021]:=50.300;
	stepTestFull[2022]:=50.300;
	stepTestFull[2023]:=50.300;
	stepTestFull[2024]:=50.300;
	stepTestFull[2025]:=50.300;
	stepTestFull[2026]:=50.300;
	stepTestFull[2027]:=50.300;
	stepTestFull[2028]:=50.300;
	stepTestFull[2029]:=50.300;
	stepTestFull[2030]:=50.300;
	stepTestFull[2031]:=50.300;
	stepTestFull[2032]:=50.300;
	stepTestFull[2033]:=50.300;
	stepTestFull[2034]:=50.300;
	stepTestFull[2035]:=50.300;
	stepTestFull[2036]:=50.300;
	stepTestFull[2037]:=50.300;
	stepTestFull[2038]:=50.300;
	stepTestFull[2039]:=50.300;
	stepTestFull[2040]:=50.300;
	stepTestFull[2041]:=50.300;
	stepTestFull[2042]:=50.300;
	stepTestFull[2043]:=50.300;
	stepTestFull[2044]:=50.300;
	stepTestFull[2045]:=50.300;
	stepTestFull[2046]:=50.300;
	stepTestFull[2047]:=50.300;
	stepTestFull[2048]:=50.300;
	stepTestFull[2049]:=50.300;
	stepTestFull[2050]:=50.300;
	stepTestFull[2051]:=50.300;
	stepTestFull[2052]:=50.300;
	stepTestFull[2053]:=50.300;
	stepTestFull[2054]:=50.300;
	stepTestFull[2055]:=50.300;
	stepTestFull[2056]:=50.300;
	stepTestFull[2057]:=50.300;
	stepTestFull[2058]:=50.300;
	stepTestFull[2059]:=50.300;
	stepTestFull[2060]:=50.300;
	stepTestFull[2061]:=50.300;
	stepTestFull[2062]:=50.300;
	stepTestFull[2063]:=50.300;
	stepTestFull[2064]:=50.300;
	stepTestFull[2065]:=50.300;
	stepTestFull[2066]:=50.300;
	stepTestFull[2067]:=50.300;
	stepTestFull[2068]:=50.300;
	stepTestFull[2069]:=50.300;
	stepTestFull[2070]:=50.300;
	stepTestFull[2071]:=50.300;
	stepTestFull[2072]:=50.300;
	stepTestFull[2073]:=50.300;
	stepTestFull[2074]:=50.300;
	stepTestFull[2075]:=50.300;
	stepTestFull[2076]:=50.300;
	stepTestFull[2077]:=50.300;
	stepTestFull[2078]:=50.300;
	stepTestFull[2079]:=50.300;
	stepTestFull[2080]:=50.300;
	stepTestFull[2081]:=50.300;
	stepTestFull[2082]:=50.300;
	stepTestFull[2083]:=50.300;
	stepTestFull[2084]:=50.300;
	stepTestFull[2085]:=50.300;
	stepTestFull[2086]:=50.300;
	stepTestFull[2087]:=50.300;
	stepTestFull[2088]:=50.300;
	stepTestFull[2089]:=50.300;
	stepTestFull[2090]:=50.300;
	stepTestFull[2091]:=50.300;
	stepTestFull[2092]:=50.300;
	stepTestFull[2093]:=50.300;
	stepTestFull[2094]:=50.300;
	stepTestFull[2095]:=50.300;
	stepTestFull[2096]:=50.300;
	stepTestFull[2097]:=50.300;
	stepTestFull[2098]:=50.300;
	stepTestFull[2099]:=50.300;
	stepTestFull[2100]:=50.300;
	stepTestFull[2101]:=50.300;
	stepTestFull[2102]:=50.300;
	stepTestFull[2103]:=50.300;
	stepTestFull[2104]:=50.300;
	stepTestFull[2105]:=50.300;
	stepTestFull[2106]:=50.300;
	stepTestFull[2107]:=50.300;
	stepTestFull[2108]:=50.300;
	stepTestFull[2109]:=50.300;
	stepTestFull[2110]:=50.300;
	stepTestFull[2111]:=50.300;
	stepTestFull[2112]:=50.300;
	stepTestFull[2113]:=50.300;
	stepTestFull[2114]:=50.300;
	stepTestFull[2115]:=50.300;
	stepTestFull[2116]:=50.300;
	stepTestFull[2117]:=50.300;
	stepTestFull[2118]:=50.300;
	stepTestFull[2119]:=50.300;
	stepTestFull[2120]:=50.300;
	stepTestFull[2121]:=50.300;
	stepTestFull[2122]:=50.300;
	stepTestFull[2123]:=50.300;
	stepTestFull[2124]:=50.300;
	stepTestFull[2125]:=50.300;
	stepTestFull[2126]:=50.300;
	stepTestFull[2127]:=50.300;
	stepTestFull[2128]:=50.300;
	stepTestFull[2129]:=50.300;
	stepTestFull[2130]:=50.000;
	stepTestFull[2131]:=50.000;
	stepTestFull[2132]:=50.000;
	stepTestFull[2133]:=50.000;
	stepTestFull[2134]:=50.000;
	stepTestFull[2135]:=50.000;
	stepTestFull[2136]:=50.000;
	stepTestFull[2137]:=50.000;
	stepTestFull[2138]:=50.000;
	stepTestFull[2139]:=50.000;
	stepTestFull[2140]:=50.000;
	stepTestFull[2141]:=50.000;
	stepTestFull[2142]:=50.000;
	stepTestFull[2143]:=50.000;
	stepTestFull[2144]:=50.000;
	stepTestFull[2145]:=50.000;
	stepTestFull[2146]:=50.000;
	stepTestFull[2147]:=50.000;
	stepTestFull[2148]:=50.000;
	stepTestFull[2149]:=50.000;
	stepTestFull[2150]:=50.000;
	stepTestFull[2151]:=50.000;
	stepTestFull[2152]:=50.000;
	stepTestFull[2153]:=50.000;
	stepTestFull[2154]:=50.000;
	stepTestFull[2155]:=50.000;
	stepTestFull[2156]:=50.000;
	stepTestFull[2157]:=50.000;
	stepTestFull[2158]:=50.000;
	stepTestFull[2159]:=50.000;
	stepTestFull[2160]:=50.000;
	stepTestFull[2161]:=50.000;
	stepTestFull[2162]:=50.000;
	stepTestFull[2163]:=50.000;
	stepTestFull[2164]:=50.000;
	stepTestFull[2165]:=50.000;
	stepTestFull[2166]:=50.000;
	stepTestFull[2167]:=50.000;
	stepTestFull[2168]:=50.000;
	stepTestFull[2169]:=50.000;
	stepTestFull[2170]:=50.000;
	stepTestFull[2171]:=50.000;
	stepTestFull[2172]:=50.000;
	stepTestFull[2173]:=50.000;
	stepTestFull[2174]:=50.000;
	stepTestFull[2175]:=50.000;
	stepTestFull[2176]:=50.000;
	stepTestFull[2177]:=50.000;
	stepTestFull[2178]:=50.000;
	stepTestFull[2179]:=50.000;
	stepTestFull[2180]:=50.000;
	stepTestFull[2181]:=50.000;
	stepTestFull[2182]:=50.000;
	stepTestFull[2183]:=50.000;
	stepTestFull[2184]:=50.000;
	stepTestFull[2185]:=50.000;
	stepTestFull[2186]:=50.000;
	stepTestFull[2187]:=50.000;
	stepTestFull[2188]:=50.000;
	stepTestFull[2189]:=50.000;
	stepTestFull[2190]:=49.700;
	stepTestFull[2191]:=49.700;
	stepTestFull[2192]:=49.700;
	stepTestFull[2193]:=49.700;
	stepTestFull[2194]:=49.700;
	stepTestFull[2195]:=49.700;
	stepTestFull[2196]:=49.700;
	stepTestFull[2197]:=49.700;
	stepTestFull[2198]:=49.700;
	stepTestFull[2199]:=49.700;
	stepTestFull[2200]:=49.700;
	stepTestFull[2201]:=49.700;
	stepTestFull[2202]:=49.700;
	stepTestFull[2203]:=49.700;
	stepTestFull[2204]:=49.700;
	stepTestFull[2205]:=49.700;
	stepTestFull[2206]:=49.700;
	stepTestFull[2207]:=49.700;
	stepTestFull[2208]:=49.700;
	stepTestFull[2209]:=49.700;
	stepTestFull[2210]:=49.700;
	stepTestFull[2211]:=49.700;
	stepTestFull[2212]:=49.700;
	stepTestFull[2213]:=49.700;
	stepTestFull[2214]:=49.700;
	stepTestFull[2215]:=49.700;
	stepTestFull[2216]:=49.700;
	stepTestFull[2217]:=49.700;
	stepTestFull[2218]:=49.700;
	stepTestFull[2219]:=49.700;
	stepTestFull[2220]:=49.700;
	stepTestFull[2221]:=49.700;
	stepTestFull[2222]:=49.700;
	stepTestFull[2223]:=49.700;
	stepTestFull[2224]:=49.700;
	stepTestFull[2225]:=49.700;
	stepTestFull[2226]:=49.700;
	stepTestFull[2227]:=49.700;
	stepTestFull[2228]:=49.700;
	stepTestFull[2229]:=49.700;
	stepTestFull[2230]:=49.700;
	stepTestFull[2231]:=49.700;
	stepTestFull[2232]:=49.700;
	stepTestFull[2233]:=49.700;
	stepTestFull[2234]:=49.700;
	stepTestFull[2235]:=49.700;
	stepTestFull[2236]:=49.700;
	stepTestFull[2237]:=49.700;
	stepTestFull[2238]:=49.700;
	stepTestFull[2239]:=49.700;
	stepTestFull[2240]:=49.700;
	stepTestFull[2241]:=49.700;
	stepTestFull[2242]:=49.700;
	stepTestFull[2243]:=49.700;
	stepTestFull[2244]:=49.700;
	stepTestFull[2245]:=49.700;
	stepTestFull[2246]:=49.700;
	stepTestFull[2247]:=49.700;
	stepTestFull[2248]:=49.700;
	stepTestFull[2249]:=49.700;
	stepTestFull[2250]:=49.700;
	stepTestFull[2251]:=49.700;
	stepTestFull[2252]:=49.700;
	stepTestFull[2253]:=49.700;
	stepTestFull[2254]:=49.700;
	stepTestFull[2255]:=49.700;
	stepTestFull[2256]:=49.700;
	stepTestFull[2257]:=49.700;
	stepTestFull[2258]:=49.700;
	stepTestFull[2259]:=49.700;
	stepTestFull[2260]:=49.700;
	stepTestFull[2261]:=49.700;
	stepTestFull[2262]:=49.700;
	stepTestFull[2263]:=49.700;
	stepTestFull[2264]:=49.700;
	stepTestFull[2265]:=49.700;
	stepTestFull[2266]:=49.700;
	stepTestFull[2267]:=49.700;
	stepTestFull[2268]:=49.700;
	stepTestFull[2269]:=49.700;
	stepTestFull[2270]:=49.700;
	stepTestFull[2271]:=49.700;
	stepTestFull[2272]:=49.700;
	stepTestFull[2273]:=49.700;
	stepTestFull[2274]:=49.700;
	stepTestFull[2275]:=49.700;
	stepTestFull[2276]:=49.700;
	stepTestFull[2277]:=49.700;
	stepTestFull[2278]:=49.700;
	stepTestFull[2279]:=49.700;
	stepTestFull[2280]:=49.700;
	stepTestFull[2281]:=49.700;
	stepTestFull[2282]:=49.700;
	stepTestFull[2283]:=49.700;
	stepTestFull[2284]:=49.700;
	stepTestFull[2285]:=49.700;
	stepTestFull[2286]:=49.700;
	stepTestFull[2287]:=49.700;
	stepTestFull[2288]:=49.700;
	stepTestFull[2289]:=49.700;
	stepTestFull[2290]:=49.700;
	stepTestFull[2291]:=49.700;
	stepTestFull[2292]:=49.700;
	stepTestFull[2293]:=49.700;
	stepTestFull[2294]:=49.700;
	stepTestFull[2295]:=49.700;
	stepTestFull[2296]:=49.700;
	stepTestFull[2297]:=49.700;
	stepTestFull[2298]:=49.700;
	stepTestFull[2299]:=49.700;
	stepTestFull[2300]:=49.700;
	stepTestFull[2301]:=49.700;
	stepTestFull[2302]:=49.700;
	stepTestFull[2303]:=49.700;
	stepTestFull[2304]:=49.700;
	stepTestFull[2305]:=49.700;
	stepTestFull[2306]:=49.700;
	stepTestFull[2307]:=49.700;
	stepTestFull[2308]:=49.700;
	stepTestFull[2309]:=49.700;
	stepTestFull[2310]:=49.700;
	stepTestFull[2311]:=49.700;
	stepTestFull[2312]:=49.700;
	stepTestFull[2313]:=49.700;
	stepTestFull[2314]:=49.700;
	stepTestFull[2315]:=49.700;
	stepTestFull[2316]:=49.700;
	stepTestFull[2317]:=49.700;
	stepTestFull[2318]:=49.700;
	stepTestFull[2319]:=49.700;
	stepTestFull[2320]:=49.700;
	stepTestFull[2321]:=49.700;
	stepTestFull[2322]:=49.700;
	stepTestFull[2323]:=49.700;
	stepTestFull[2324]:=49.700;
	stepTestFull[2325]:=49.700;
	stepTestFull[2326]:=49.700;
	stepTestFull[2327]:=49.700;
	stepTestFull[2328]:=49.700;
	stepTestFull[2329]:=49.700;
	stepTestFull[2330]:=49.700;
	stepTestFull[2331]:=49.700;
	stepTestFull[2332]:=49.700;
	stepTestFull[2333]:=49.700;
	stepTestFull[2334]:=49.700;
	stepTestFull[2335]:=49.700;
	stepTestFull[2336]:=49.700;
	stepTestFull[2337]:=49.700;
	stepTestFull[2338]:=49.700;
	stepTestFull[2339]:=49.700;
	stepTestFull[2340]:=49.700;
	stepTestFull[2341]:=49.700;
	stepTestFull[2342]:=49.700;
	stepTestFull[2343]:=49.700;
	stepTestFull[2344]:=49.700;
	stepTestFull[2345]:=49.700;
	stepTestFull[2346]:=49.700;
	stepTestFull[2347]:=49.700;
	stepTestFull[2348]:=49.700;
	stepTestFull[2349]:=49.700;
	stepTestFull[2350]:=49.700;
	stepTestFull[2351]:=49.700;
	stepTestFull[2352]:=49.700;
	stepTestFull[2353]:=49.700;
	stepTestFull[2354]:=49.700;
	stepTestFull[2355]:=49.700;
	stepTestFull[2356]:=49.700;
	stepTestFull[2357]:=49.700;
	stepTestFull[2358]:=49.700;
	stepTestFull[2359]:=49.700;
	stepTestFull[2360]:=49.700;
	stepTestFull[2361]:=49.700;
	stepTestFull[2362]:=49.700;
	stepTestFull[2363]:=49.700;
	stepTestFull[2364]:=49.700;
	stepTestFull[2365]:=49.700;
	stepTestFull[2366]:=49.700;
	stepTestFull[2367]:=49.700;
	stepTestFull[2368]:=49.700;
	stepTestFull[2369]:=49.700;
	stepTestFull[2370]:=50.000;
	stepTestFull[2371]:=50.000;
	stepTestFull[2372]:=50.000;
	stepTestFull[2373]:=50.000;
	stepTestFull[2374]:=50.000;
	stepTestFull[2375]:=50.000;
	stepTestFull[2376]:=50.000;
	stepTestFull[2377]:=50.000;
	stepTestFull[2378]:=50.000;
	stepTestFull[2379]:=50.000;
	stepTestFull[2380]:=50.000;
	stepTestFull[2381]:=50.000;
	stepTestFull[2382]:=50.000;
	stepTestFull[2383]:=50.000;
	stepTestFull[2384]:=50.000;
	stepTestFull[2385]:=50.000;
	stepTestFull[2386]:=50.000;
	stepTestFull[2387]:=50.000;
	stepTestFull[2388]:=50.000;
	stepTestFull[2389]:=50.000;
	stepTestFull[2390]:=50.000;
	stepTestFull[2391]:=50.000;
	stepTestFull[2392]:=50.000;
	stepTestFull[2393]:=50.000;
	stepTestFull[2394]:=50.000;
	stepTestFull[2395]:=50.000;
	stepTestFull[2396]:=50.000;
	stepTestFull[2397]:=50.000;
	stepTestFull[2398]:=50.000;
	stepTestFull[2399]:=50.000;
	stepTestFull[2400]:=50.000;
	stepTestFull[2401]:=50.000;
	stepTestFull[2402]:=50.000;
	stepTestFull[2403]:=50.000;
	stepTestFull[2404]:=50.000;
	stepTestFull[2405]:=50.000;
	stepTestFull[2406]:=50.000;
	stepTestFull[2407]:=50.000;
	stepTestFull[2408]:=50.000;
	stepTestFull[2409]:=50.000;
	stepTestFull[2410]:=50.000;
	stepTestFull[2411]:=50.000;
	stepTestFull[2412]:=50.000;
	stepTestFull[2413]:=50.000;
	stepTestFull[2414]:=50.000;
	stepTestFull[2415]:=50.000;
	stepTestFull[2416]:=50.000;
	stepTestFull[2417]:=50.000;
	stepTestFull[2418]:=50.000;
	stepTestFull[2419]:=50.000;
	stepTestFull[2420]:=50.000;
	stepTestFull[2421]:=50.000;
	stepTestFull[2422]:=50.000;
	stepTestFull[2423]:=50.000;
	stepTestFull[2424]:=50.000;
	stepTestFull[2425]:=50.000;
	stepTestFull[2426]:=50.000;
	stepTestFull[2427]:=50.000;
	stepTestFull[2428]:=50.000;
	stepTestFull[2429]:=50.000;
	stepTestFull[2430]:=50.400;
	stepTestFull[2431]:=50.400;
	stepTestFull[2432]:=50.400;
	stepTestFull[2433]:=50.400;
	stepTestFull[2434]:=50.400;
	stepTestFull[2435]:=50.400;
	stepTestFull[2436]:=50.400;
	stepTestFull[2437]:=50.400;
	stepTestFull[2438]:=50.400;
	stepTestFull[2439]:=50.400;
	stepTestFull[2440]:=50.400;
	stepTestFull[2441]:=50.400;
	stepTestFull[2442]:=50.400;
	stepTestFull[2443]:=50.400;
	stepTestFull[2444]:=50.400;
	stepTestFull[2445]:=50.400;
	stepTestFull[2446]:=50.400;
	stepTestFull[2447]:=50.400;
	stepTestFull[2448]:=50.400;
	stepTestFull[2449]:=50.400;
	stepTestFull[2450]:=50.400;
	stepTestFull[2451]:=50.400;
	stepTestFull[2452]:=50.400;
	stepTestFull[2453]:=50.400;
	stepTestFull[2454]:=50.400;
	stepTestFull[2455]:=50.400;
	stepTestFull[2456]:=50.400;
	stepTestFull[2457]:=50.400;
	stepTestFull[2458]:=50.400;
	stepTestFull[2459]:=50.400;
	stepTestFull[2460]:=50.400;
	stepTestFull[2461]:=50.400;
	stepTestFull[2462]:=50.400;
	stepTestFull[2463]:=50.400;
	stepTestFull[2464]:=50.400;
	stepTestFull[2465]:=50.400;
	stepTestFull[2466]:=50.400;
	stepTestFull[2467]:=50.400;
	stepTestFull[2468]:=50.400;
	stepTestFull[2469]:=50.400;
	stepTestFull[2470]:=50.400;
	stepTestFull[2471]:=50.400;
	stepTestFull[2472]:=50.400;
	stepTestFull[2473]:=50.400;
	stepTestFull[2474]:=50.400;
	stepTestFull[2475]:=50.400;
	stepTestFull[2476]:=50.400;
	stepTestFull[2477]:=50.400;
	stepTestFull[2478]:=50.400;
	stepTestFull[2479]:=50.400;
	stepTestFull[2480]:=50.400;
	stepTestFull[2481]:=50.400;
	stepTestFull[2482]:=50.400;
	stepTestFull[2483]:=50.400;
	stepTestFull[2484]:=50.400;
	stepTestFull[2485]:=50.400;
	stepTestFull[2486]:=50.400;
	stepTestFull[2487]:=50.400;
	stepTestFull[2488]:=50.400;
	stepTestFull[2489]:=50.400;
	stepTestFull[2490]:=50.400;
	stepTestFull[2491]:=50.400;
	stepTestFull[2492]:=50.400;
	stepTestFull[2493]:=50.400;
	stepTestFull[2494]:=50.400;
	stepTestFull[2495]:=50.400;
	stepTestFull[2496]:=50.400;
	stepTestFull[2497]:=50.400;
	stepTestFull[2498]:=50.400;
	stepTestFull[2499]:=50.400;
	stepTestFull[2500]:=50.400;
	stepTestFull[2501]:=50.400;
	stepTestFull[2502]:=50.400;
	stepTestFull[2503]:=50.400;
	stepTestFull[2504]:=50.400;
	stepTestFull[2505]:=50.400;
	stepTestFull[2506]:=50.400;
	stepTestFull[2507]:=50.400;
	stepTestFull[2508]:=50.400;
	stepTestFull[2509]:=50.400;
	stepTestFull[2510]:=50.400;
	stepTestFull[2511]:=50.400;
	stepTestFull[2512]:=50.400;
	stepTestFull[2513]:=50.400;
	stepTestFull[2514]:=50.400;
	stepTestFull[2515]:=50.400;
	stepTestFull[2516]:=50.400;
	stepTestFull[2517]:=50.400;
	stepTestFull[2518]:=50.400;
	stepTestFull[2519]:=50.400;
	stepTestFull[2520]:=50.400;
	stepTestFull[2521]:=50.400;
	stepTestFull[2522]:=50.400;
	stepTestFull[2523]:=50.400;
	stepTestFull[2524]:=50.400;
	stepTestFull[2525]:=50.400;
	stepTestFull[2526]:=50.400;
	stepTestFull[2527]:=50.400;
	stepTestFull[2528]:=50.400;
	stepTestFull[2529]:=50.400;
	stepTestFull[2530]:=50.400;
	stepTestFull[2531]:=50.400;
	stepTestFull[2532]:=50.400;
	stepTestFull[2533]:=50.400;
	stepTestFull[2534]:=50.400;
	stepTestFull[2535]:=50.400;
	stepTestFull[2536]:=50.400;
	stepTestFull[2537]:=50.400;
	stepTestFull[2538]:=50.400;
	stepTestFull[2539]:=50.400;
	stepTestFull[2540]:=50.400;
	stepTestFull[2541]:=50.400;
	stepTestFull[2542]:=50.400;
	stepTestFull[2543]:=50.400;
	stepTestFull[2544]:=50.400;
	stepTestFull[2545]:=50.400;
	stepTestFull[2546]:=50.400;
	stepTestFull[2547]:=50.400;
	stepTestFull[2548]:=50.400;
	stepTestFull[2549]:=50.400;
	stepTestFull[2550]:=50.400;
	stepTestFull[2551]:=50.400;
	stepTestFull[2552]:=50.400;
	stepTestFull[2553]:=50.400;
	stepTestFull[2554]:=50.400;
	stepTestFull[2555]:=50.400;
	stepTestFull[2556]:=50.400;
	stepTestFull[2557]:=50.400;
	stepTestFull[2558]:=50.400;
	stepTestFull[2559]:=50.400;
	stepTestFull[2560]:=50.400;
	stepTestFull[2561]:=50.400;
	stepTestFull[2562]:=50.400;
	stepTestFull[2563]:=50.400;
	stepTestFull[2564]:=50.400;
	stepTestFull[2565]:=50.400;
	stepTestFull[2566]:=50.400;
	stepTestFull[2567]:=50.400;
	stepTestFull[2568]:=50.400;
	stepTestFull[2569]:=50.400;
	stepTestFull[2570]:=50.400;
	stepTestFull[2571]:=50.400;
	stepTestFull[2572]:=50.400;
	stepTestFull[2573]:=50.400;
	stepTestFull[2574]:=50.400;
	stepTestFull[2575]:=50.400;
	stepTestFull[2576]:=50.400;
	stepTestFull[2577]:=50.400;
	stepTestFull[2578]:=50.400;
	stepTestFull[2579]:=50.400;
	stepTestFull[2580]:=50.400;
	stepTestFull[2581]:=50.400;
	stepTestFull[2582]:=50.400;
	stepTestFull[2583]:=50.400;
	stepTestFull[2584]:=50.400;
	stepTestFull[2585]:=50.400;
	stepTestFull[2586]:=50.400;
	stepTestFull[2587]:=50.400;
	stepTestFull[2588]:=50.400;
	stepTestFull[2589]:=50.400;
	stepTestFull[2590]:=50.400;
	stepTestFull[2591]:=50.400;
	stepTestFull[2592]:=50.400;
	stepTestFull[2593]:=50.400;
	stepTestFull[2594]:=50.400;
	stepTestFull[2595]:=50.400;
	stepTestFull[2596]:=50.400;
	stepTestFull[2597]:=50.400;
	stepTestFull[2598]:=50.400;
	stepTestFull[2599]:=50.400;
	stepTestFull[2600]:=50.400;
	stepTestFull[2601]:=50.400;
	stepTestFull[2602]:=50.400;
	stepTestFull[2603]:=50.400;
	stepTestFull[2604]:=50.400;
	stepTestFull[2605]:=50.400;
	stepTestFull[2606]:=50.400;
	stepTestFull[2607]:=50.400;
	stepTestFull[2608]:=50.400;
	stepTestFull[2609]:=50.400;
	stepTestFull[2610]:=50.000;
	stepTestFull[2611]:=50.000;
	stepTestFull[2612]:=50.000;
	stepTestFull[2613]:=50.000;
	stepTestFull[2614]:=50.000;
	stepTestFull[2615]:=50.000;
	stepTestFull[2616]:=50.000;
	stepTestFull[2617]:=50.000;
	stepTestFull[2618]:=50.000;
	stepTestFull[2619]:=50.000;
	stepTestFull[2620]:=50.000;
	stepTestFull[2621]:=50.000;
	stepTestFull[2622]:=50.000;
	stepTestFull[2623]:=50.000;
	stepTestFull[2624]:=50.000;
	stepTestFull[2625]:=50.000;
	stepTestFull[2626]:=50.000;
	stepTestFull[2627]:=50.000;
	stepTestFull[2628]:=50.000;
	stepTestFull[2629]:=50.000;
	stepTestFull[2630]:=50.000;
	stepTestFull[2631]:=50.000;
	stepTestFull[2632]:=50.000;
	stepTestFull[2633]:=50.000;
	stepTestFull[2634]:=50.000;
	stepTestFull[2635]:=50.000;
	stepTestFull[2636]:=50.000;
	stepTestFull[2637]:=50.000;
	stepTestFull[2638]:=50.000;
	stepTestFull[2639]:=50.000;
	stepTestFull[2640]:=50.000;
	stepTestFull[2641]:=50.000;
	stepTestFull[2642]:=50.000;
	stepTestFull[2643]:=50.000;
	stepTestFull[2644]:=50.000;
	stepTestFull[2645]:=50.000;
	stepTestFull[2646]:=50.000;
	stepTestFull[2647]:=50.000;
	stepTestFull[2648]:=50.000;
	stepTestFull[2649]:=50.000;
	stepTestFull[2650]:=50.000;
	stepTestFull[2651]:=50.000;
	stepTestFull[2652]:=50.000;
	stepTestFull[2653]:=50.000;
	stepTestFull[2654]:=50.000;
	stepTestFull[2655]:=50.000;
	stepTestFull[2656]:=50.000;
	stepTestFull[2657]:=50.000;
	stepTestFull[2658]:=50.000;
	stepTestFull[2659]:=50.000;
	stepTestFull[2660]:=50.000;
	stepTestFull[2661]:=50.000;
	stepTestFull[2662]:=50.000;
	stepTestFull[2663]:=50.000;
	stepTestFull[2664]:=50.000;
	stepTestFull[2665]:=50.000;
	stepTestFull[2666]:=50.000;
	stepTestFull[2667]:=50.000;
	stepTestFull[2668]:=50.000;
	stepTestFull[2669]:=50.000;
	stepTestFull[2670]:=49.600;
	stepTestFull[2671]:=49.600;
	stepTestFull[2672]:=49.600;
	stepTestFull[2673]:=49.600;
	stepTestFull[2674]:=49.600;
	stepTestFull[2675]:=49.600;
	stepTestFull[2676]:=49.600;
	stepTestFull[2677]:=49.600;
	stepTestFull[2678]:=49.600;
	stepTestFull[2679]:=49.600;
	stepTestFull[2680]:=49.600;
	stepTestFull[2681]:=49.600;
	stepTestFull[2682]:=49.600;
	stepTestFull[2683]:=49.600;
	stepTestFull[2684]:=49.600;
	stepTestFull[2685]:=49.600;
	stepTestFull[2686]:=49.600;
	stepTestFull[2687]:=49.600;
	stepTestFull[2688]:=49.600;
	stepTestFull[2689]:=49.600;
	stepTestFull[2690]:=49.600;
	stepTestFull[2691]:=49.600;
	stepTestFull[2692]:=49.600;
	stepTestFull[2693]:=49.600;
	stepTestFull[2694]:=49.600;
	stepTestFull[2695]:=49.600;
	stepTestFull[2696]:=49.600;
	stepTestFull[2697]:=49.600;
	stepTestFull[2698]:=49.600;
	stepTestFull[2699]:=49.600;
	stepTestFull[2700]:=49.600;
	stepTestFull[2701]:=49.600;
	stepTestFull[2702]:=49.600;
	stepTestFull[2703]:=49.600;
	stepTestFull[2704]:=49.600;
	stepTestFull[2705]:=49.600;
	stepTestFull[2706]:=49.600;
	stepTestFull[2707]:=49.600;
	stepTestFull[2708]:=49.600;
	stepTestFull[2709]:=49.600;
	stepTestFull[2710]:=49.600;
	stepTestFull[2711]:=49.600;
	stepTestFull[2712]:=49.600;
	stepTestFull[2713]:=49.600;
	stepTestFull[2714]:=49.600;
	stepTestFull[2715]:=49.600;
	stepTestFull[2716]:=49.600;
	stepTestFull[2717]:=49.600;
	stepTestFull[2718]:=49.600;
	stepTestFull[2719]:=49.600;
	stepTestFull[2720]:=49.600;
	stepTestFull[2721]:=49.600;
	stepTestFull[2722]:=49.600;
	stepTestFull[2723]:=49.600;
	stepTestFull[2724]:=49.600;
	stepTestFull[2725]:=49.600;
	stepTestFull[2726]:=49.600;
	stepTestFull[2727]:=49.600;
	stepTestFull[2728]:=49.600;
	stepTestFull[2729]:=49.600;
	stepTestFull[2730]:=49.600;
	stepTestFull[2731]:=49.600;
	stepTestFull[2732]:=49.600;
	stepTestFull[2733]:=49.600;
	stepTestFull[2734]:=49.600;
	stepTestFull[2735]:=49.600;
	stepTestFull[2736]:=49.600;
	stepTestFull[2737]:=49.600;
	stepTestFull[2738]:=49.600;
	stepTestFull[2739]:=49.600;
	stepTestFull[2740]:=49.600;
	stepTestFull[2741]:=49.600;
	stepTestFull[2742]:=49.600;
	stepTestFull[2743]:=49.600;
	stepTestFull[2744]:=49.600;
	stepTestFull[2745]:=49.600;
	stepTestFull[2746]:=49.600;
	stepTestFull[2747]:=49.600;
	stepTestFull[2748]:=49.600;
	stepTestFull[2749]:=49.600;
	stepTestFull[2750]:=49.600;
	stepTestFull[2751]:=49.600;
	stepTestFull[2752]:=49.600;
	stepTestFull[2753]:=49.600;
	stepTestFull[2754]:=49.600;
	stepTestFull[2755]:=49.600;
	stepTestFull[2756]:=49.600;
	stepTestFull[2757]:=49.600;
	stepTestFull[2758]:=49.600;
	stepTestFull[2759]:=49.600;
	stepTestFull[2760]:=49.600;
	stepTestFull[2761]:=49.600;
	stepTestFull[2762]:=49.600;
	stepTestFull[2763]:=49.600;
	stepTestFull[2764]:=49.600;
	stepTestFull[2765]:=49.600;
	stepTestFull[2766]:=49.600;
	stepTestFull[2767]:=49.600;
	stepTestFull[2768]:=49.600;
	stepTestFull[2769]:=49.600;
	stepTestFull[2770]:=49.600;
	stepTestFull[2771]:=49.600;
	stepTestFull[2772]:=49.600;
	stepTestFull[2773]:=49.600;
	stepTestFull[2774]:=49.600;
	stepTestFull[2775]:=49.600;
	stepTestFull[2776]:=49.600;
	stepTestFull[2777]:=49.600;
	stepTestFull[2778]:=49.600;
	stepTestFull[2779]:=49.600;
	stepTestFull[2780]:=49.600;
	stepTestFull[2781]:=49.600;
	stepTestFull[2782]:=49.600;
	stepTestFull[2783]:=49.600;
	stepTestFull[2784]:=49.600;
	stepTestFull[2785]:=49.600;
	stepTestFull[2786]:=49.600;
	stepTestFull[2787]:=49.600;
	stepTestFull[2788]:=49.600;
	stepTestFull[2789]:=49.600;
	stepTestFull[2790]:=49.600;
	stepTestFull[2791]:=49.600;
	stepTestFull[2792]:=49.600;
	stepTestFull[2793]:=49.600;
	stepTestFull[2794]:=49.600;
	stepTestFull[2795]:=49.600;
	stepTestFull[2796]:=49.600;
	stepTestFull[2797]:=49.600;
	stepTestFull[2798]:=49.600;
	stepTestFull[2799]:=49.600;
	stepTestFull[2800]:=49.600;
	stepTestFull[2801]:=49.600;
	stepTestFull[2802]:=49.600;
	stepTestFull[2803]:=49.600;
	stepTestFull[2804]:=49.600;
	stepTestFull[2805]:=49.600;
	stepTestFull[2806]:=49.600;
	stepTestFull[2807]:=49.600;
	stepTestFull[2808]:=49.600;
	stepTestFull[2809]:=49.600;
	stepTestFull[2810]:=49.600;
	stepTestFull[2811]:=49.600;
	stepTestFull[2812]:=49.600;
	stepTestFull[2813]:=49.600;
	stepTestFull[2814]:=49.600;
	stepTestFull[2815]:=49.600;
	stepTestFull[2816]:=49.600;
	stepTestFull[2817]:=49.600;
	stepTestFull[2818]:=49.600;
	stepTestFull[2819]:=49.600;
	stepTestFull[2820]:=49.600;
	stepTestFull[2821]:=49.600;
	stepTestFull[2822]:=49.600;
	stepTestFull[2823]:=49.600;
	stepTestFull[2824]:=49.600;
	stepTestFull[2825]:=49.600;
	stepTestFull[2826]:=49.600;
	stepTestFull[2827]:=49.600;
	stepTestFull[2828]:=49.600;
	stepTestFull[2829]:=49.600;
	stepTestFull[2830]:=49.600;
	stepTestFull[2831]:=49.600;
	stepTestFull[2832]:=49.600;
	stepTestFull[2833]:=49.600;
	stepTestFull[2834]:=49.600;
	stepTestFull[2835]:=49.600;
	stepTestFull[2836]:=49.600;
	stepTestFull[2837]:=49.600;
	stepTestFull[2838]:=49.600;
	stepTestFull[2839]:=49.600;
	stepTestFull[2840]:=49.600;
	stepTestFull[2841]:=49.600;
	stepTestFull[2842]:=49.600;
	stepTestFull[2843]:=49.600;
	stepTestFull[2844]:=49.600;
	stepTestFull[2845]:=49.600;
	stepTestFull[2846]:=49.600;
	stepTestFull[2847]:=49.600;
	stepTestFull[2848]:=49.600;
	stepTestFull[2849]:=49.600;
	stepTestFull[2850]:=50.000;
	stepTestFull[2851]:=50.000;
	stepTestFull[2852]:=50.000;
	stepTestFull[2853]:=50.000;
	stepTestFull[2854]:=50.000;
	stepTestFull[2855]:=50.000;
	stepTestFull[2856]:=50.000;
	stepTestFull[2857]:=50.000;
	stepTestFull[2858]:=50.000;
	stepTestFull[2859]:=50.000;
	stepTestFull[2860]:=50.000;
	stepTestFull[2861]:=50.000;
	stepTestFull[2862]:=50.000;
	stepTestFull[2863]:=50.000;
	stepTestFull[2864]:=50.000;
	stepTestFull[2865]:=50.000;
	stepTestFull[2866]:=50.000;
	stepTestFull[2867]:=50.000;
	stepTestFull[2868]:=50.000;
	stepTestFull[2869]:=50.000;
	stepTestFull[2870]:=50.000;
	stepTestFull[2871]:=50.000;
	stepTestFull[2872]:=50.000;
	stepTestFull[2873]:=50.000;
	stepTestFull[2874]:=50.000;
	stepTestFull[2875]:=50.000;
	stepTestFull[2876]:=50.000;
	stepTestFull[2877]:=50.000;
	stepTestFull[2878]:=50.000;
	stepTestFull[2879]:=50.000;
	stepTestFull[2880]:=50.000;
	stepTestFull[2881]:=50.000;
	stepTestFull[2882]:=50.000;
	stepTestFull[2883]:=50.000;
	stepTestFull[2884]:=50.000;
	stepTestFull[2885]:=50.000;
	stepTestFull[2886]:=50.000;
	stepTestFull[2887]:=50.000;
	stepTestFull[2888]:=50.000;
	stepTestFull[2889]:=50.000;
	stepTestFull[2890]:=50.000;
	stepTestFull[2891]:=50.000;
	stepTestFull[2892]:=50.000;
	stepTestFull[2893]:=50.000;
	stepTestFull[2894]:=50.000;
	stepTestFull[2895]:=50.000;
	stepTestFull[2896]:=50.000;
	stepTestFull[2897]:=50.000;
	stepTestFull[2898]:=50.000;
	stepTestFull[2899]:=50.000;
	stepTestFull[2900]:=50.000;
	stepTestFull[2901]:=50.000;
	stepTestFull[2902]:=50.000;
	stepTestFull[2903]:=50.000;
	stepTestFull[2904]:=50.000;
	stepTestFull[2905]:=50.000;
	stepTestFull[2906]:=50.000;
	stepTestFull[2907]:=50.000;
	stepTestFull[2908]:=50.000;
	stepTestFull[2909]:=50.000;
	stepTestFull[2910]:=50.500;
	stepTestFull[2911]:=50.500;
	stepTestFull[2912]:=50.500;
	stepTestFull[2913]:=50.500;
	stepTestFull[2914]:=50.500;
	stepTestFull[2915]:=50.500;
	stepTestFull[2916]:=50.500;
	stepTestFull[2917]:=50.500;
	stepTestFull[2918]:=50.500;
	stepTestFull[2919]:=50.500;
	stepTestFull[2920]:=50.500;
	stepTestFull[2921]:=50.500;
	stepTestFull[2922]:=50.500;
	stepTestFull[2923]:=50.500;
	stepTestFull[2924]:=50.500;
	stepTestFull[2925]:=50.500;
	stepTestFull[2926]:=50.500;
	stepTestFull[2927]:=50.500;
	stepTestFull[2928]:=50.500;
	stepTestFull[2929]:=50.500;
	stepTestFull[2930]:=50.500;
	stepTestFull[2931]:=50.500;
	stepTestFull[2932]:=50.500;
	stepTestFull[2933]:=50.500;
	stepTestFull[2934]:=50.500;
	stepTestFull[2935]:=50.500;
	stepTestFull[2936]:=50.500;
	stepTestFull[2937]:=50.500;
	stepTestFull[2938]:=50.500;
	stepTestFull[2939]:=50.500;
	stepTestFull[2940]:=50.500;
	stepTestFull[2941]:=50.500;
	stepTestFull[2942]:=50.500;
	stepTestFull[2943]:=50.500;
	stepTestFull[2944]:=50.500;
	stepTestFull[2945]:=50.500;
	stepTestFull[2946]:=50.500;
	stepTestFull[2947]:=50.500;
	stepTestFull[2948]:=50.500;
	stepTestFull[2949]:=50.500;
	stepTestFull[2950]:=50.500;
	stepTestFull[2951]:=50.500;
	stepTestFull[2952]:=50.500;
	stepTestFull[2953]:=50.500;
	stepTestFull[2954]:=50.500;
	stepTestFull[2955]:=50.500;
	stepTestFull[2956]:=50.500;
	stepTestFull[2957]:=50.500;
	stepTestFull[2958]:=50.500;
	stepTestFull[2959]:=50.500;
	stepTestFull[2960]:=50.500;
	stepTestFull[2961]:=50.500;
	stepTestFull[2962]:=50.500;
	stepTestFull[2963]:=50.500;
	stepTestFull[2964]:=50.500;
	stepTestFull[2965]:=50.500;
	stepTestFull[2966]:=50.500;
	stepTestFull[2967]:=50.500;
	stepTestFull[2968]:=50.500;
	stepTestFull[2969]:=50.500;
	stepTestFull[2970]:=50.500;
	stepTestFull[2971]:=50.500;
	stepTestFull[2972]:=50.500;
	stepTestFull[2973]:=50.500;
	stepTestFull[2974]:=50.500;
	stepTestFull[2975]:=50.500;
	stepTestFull[2976]:=50.500;
	stepTestFull[2977]:=50.500;
	stepTestFull[2978]:=50.500;
	stepTestFull[2979]:=50.500;
	stepTestFull[2980]:=50.500;
	stepTestFull[2981]:=50.500;
	stepTestFull[2982]:=50.500;
	stepTestFull[2983]:=50.500;
	stepTestFull[2984]:=50.500;
	stepTestFull[2985]:=50.500;
	stepTestFull[2986]:=50.500;
	stepTestFull[2987]:=50.500;
	stepTestFull[2988]:=50.500;
	stepTestFull[2989]:=50.500;
	stepTestFull[2990]:=50.500;
	stepTestFull[2991]:=50.500;
	stepTestFull[2992]:=50.500;
	stepTestFull[2993]:=50.500;
	stepTestFull[2994]:=50.500;
	stepTestFull[2995]:=50.500;
	stepTestFull[2996]:=50.500;
	stepTestFull[2997]:=50.500;
	stepTestFull[2998]:=50.500;
	stepTestFull[2999]:=50.500;
	stepTestFull[3000]:=50.500;
	stepTestFull[3001]:=50.500;
	stepTestFull[3002]:=50.500;
	stepTestFull[3003]:=50.500;
	stepTestFull[3004]:=50.500;
	stepTestFull[3005]:=50.500;
	stepTestFull[3006]:=50.500;
	stepTestFull[3007]:=50.500;
	stepTestFull[3008]:=50.500;
	stepTestFull[3009]:=50.500;
	stepTestFull[3010]:=50.500;
	stepTestFull[3011]:=50.500;
	stepTestFull[3012]:=50.500;
	stepTestFull[3013]:=50.500;
	stepTestFull[3014]:=50.500;
	stepTestFull[3015]:=50.500;
	stepTestFull[3016]:=50.500;
	stepTestFull[3017]:=50.500;
	stepTestFull[3018]:=50.500;
	stepTestFull[3019]:=50.500;
	stepTestFull[3020]:=50.500;
	stepTestFull[3021]:=50.500;
	stepTestFull[3022]:=50.500;
	stepTestFull[3023]:=50.500;
	stepTestFull[3024]:=50.500;
	stepTestFull[3025]:=50.500;
	stepTestFull[3026]:=50.500;
	stepTestFull[3027]:=50.500;
	stepTestFull[3028]:=50.500;
	stepTestFull[3029]:=50.500;
	stepTestFull[3030]:=50.500;
	stepTestFull[3031]:=50.500;
	stepTestFull[3032]:=50.500;
	stepTestFull[3033]:=50.500;
	stepTestFull[3034]:=50.500;
	stepTestFull[3035]:=50.500;
	stepTestFull[3036]:=50.500;
	stepTestFull[3037]:=50.500;
	stepTestFull[3038]:=50.500;
	stepTestFull[3039]:=50.500;
	stepTestFull[3040]:=50.500;
	stepTestFull[3041]:=50.500;
	stepTestFull[3042]:=50.500;
	stepTestFull[3043]:=50.500;
	stepTestFull[3044]:=50.500;
	stepTestFull[3045]:=50.500;
	stepTestFull[3046]:=50.500;
	stepTestFull[3047]:=50.500;
	stepTestFull[3048]:=50.500;
	stepTestFull[3049]:=50.500;
	stepTestFull[3050]:=50.500;
	stepTestFull[3051]:=50.500;
	stepTestFull[3052]:=50.500;
	stepTestFull[3053]:=50.500;
	stepTestFull[3054]:=50.500;
	stepTestFull[3055]:=50.500;
	stepTestFull[3056]:=50.500;
	stepTestFull[3057]:=50.500;
	stepTestFull[3058]:=50.500;
	stepTestFull[3059]:=50.500;
	stepTestFull[3060]:=50.500;
	stepTestFull[3061]:=50.500;
	stepTestFull[3062]:=50.500;
	stepTestFull[3063]:=50.500;
	stepTestFull[3064]:=50.500;
	stepTestFull[3065]:=50.500;
	stepTestFull[3066]:=50.500;
	stepTestFull[3067]:=50.500;
	stepTestFull[3068]:=50.500;
	stepTestFull[3069]:=50.500;
	stepTestFull[3070]:=50.500;
	stepTestFull[3071]:=50.500;
	stepTestFull[3072]:=50.500;
	stepTestFull[3073]:=50.500;
	stepTestFull[3074]:=50.500;
	stepTestFull[3075]:=50.500;
	stepTestFull[3076]:=50.500;
	stepTestFull[3077]:=50.500;
	stepTestFull[3078]:=50.500;
	stepTestFull[3079]:=50.500;
	stepTestFull[3080]:=50.500;
	stepTestFull[3081]:=50.500;
	stepTestFull[3082]:=50.500;
	stepTestFull[3083]:=50.500;
	stepTestFull[3084]:=50.500;
	stepTestFull[3085]:=50.500;
	stepTestFull[3086]:=50.500;
	stepTestFull[3087]:=50.500;
	stepTestFull[3088]:=50.500;
	stepTestFull[3089]:=50.500;
	stepTestFull[3090]:=50.000;
	stepTestFull[3091]:=50.000;
	stepTestFull[3092]:=50.000;
	stepTestFull[3093]:=50.000;
	stepTestFull[3094]:=50.000;
	stepTestFull[3095]:=50.000;
	stepTestFull[3096]:=50.000;
	stepTestFull[3097]:=50.000;
	stepTestFull[3098]:=50.000;
	stepTestFull[3099]:=50.000;
	stepTestFull[3100]:=50.000;
	stepTestFull[3101]:=50.000;
	stepTestFull[3102]:=50.000;
	stepTestFull[3103]:=50.000;
	stepTestFull[3104]:=50.000;
	stepTestFull[3105]:=50.000;
	stepTestFull[3106]:=50.000;
	stepTestFull[3107]:=50.000;
	stepTestFull[3108]:=50.000;
	stepTestFull[3109]:=50.000;
	stepTestFull[3110]:=50.000;
	stepTestFull[3111]:=50.000;
	stepTestFull[3112]:=50.000;
	stepTestFull[3113]:=50.000;
	stepTestFull[3114]:=50.000;
	stepTestFull[3115]:=50.000;
	stepTestFull[3116]:=50.000;
	stepTestFull[3117]:=50.000;
	stepTestFull[3118]:=50.000;
	stepTestFull[3119]:=50.000;
	stepTestFull[3120]:=50.000;
	stepTestFull[3121]:=50.000;
	stepTestFull[3122]:=50.000;
	stepTestFull[3123]:=50.000;
	stepTestFull[3124]:=50.000;
	stepTestFull[3125]:=50.000;
	stepTestFull[3126]:=50.000;
	stepTestFull[3127]:=50.000;
	stepTestFull[3128]:=50.000;
	stepTestFull[3129]:=50.000;
	stepTestFull[3130]:=50.000;
	stepTestFull[3131]:=50.000;
	stepTestFull[3132]:=50.000;
	stepTestFull[3133]:=50.000;
	stepTestFull[3134]:=50.000;
	stepTestFull[3135]:=50.000;
	stepTestFull[3136]:=50.000;
	stepTestFull[3137]:=50.000;
	stepTestFull[3138]:=50.000;
	stepTestFull[3139]:=50.000;
	stepTestFull[3140]:=50.000;
	stepTestFull[3141]:=50.000;
	stepTestFull[3142]:=50.000;
	stepTestFull[3143]:=50.000;
	stepTestFull[3144]:=50.000;
	stepTestFull[3145]:=50.000;
	stepTestFull[3146]:=50.000;
	stepTestFull[3147]:=50.000;
	stepTestFull[3148]:=50.000;
	stepTestFull[3149]:=50.000;
	stepTestFull[3150]:=49.500;
	stepTestFull[3151]:=49.500;
	stepTestFull[3152]:=49.500;
	stepTestFull[3153]:=49.500;
	stepTestFull[3154]:=49.500;
	stepTestFull[3155]:=49.500;
	stepTestFull[3156]:=49.500;
	stepTestFull[3157]:=49.500;
	stepTestFull[3158]:=49.500;
	stepTestFull[3159]:=49.500;
	stepTestFull[3160]:=49.500;
	stepTestFull[3161]:=49.500;
	stepTestFull[3162]:=49.500;
	stepTestFull[3163]:=49.500;
	stepTestFull[3164]:=49.500;
	stepTestFull[3165]:=49.500;
	stepTestFull[3166]:=49.500;
	stepTestFull[3167]:=49.500;
	stepTestFull[3168]:=49.500;
	stepTestFull[3169]:=49.500;
	stepTestFull[3170]:=49.500;
	stepTestFull[3171]:=49.500;
	stepTestFull[3172]:=49.500;
	stepTestFull[3173]:=49.500;
	stepTestFull[3174]:=49.500;
	stepTestFull[3175]:=49.500;
	stepTestFull[3176]:=49.500;
	stepTestFull[3177]:=49.500;
	stepTestFull[3178]:=49.500;
	stepTestFull[3179]:=49.500;
	stepTestFull[3180]:=49.500;
	stepTestFull[3181]:=49.500;
	stepTestFull[3182]:=49.500;
	stepTestFull[3183]:=49.500;
	stepTestFull[3184]:=49.500;
	stepTestFull[3185]:=49.500;
	stepTestFull[3186]:=49.500;
	stepTestFull[3187]:=49.500;
	stepTestFull[3188]:=49.500;
	stepTestFull[3189]:=49.500;
	stepTestFull[3190]:=49.500;
	stepTestFull[3191]:=49.500;
	stepTestFull[3192]:=49.500;
	stepTestFull[3193]:=49.500;
	stepTestFull[3194]:=49.500;
	stepTestFull[3195]:=49.500;
	stepTestFull[3196]:=49.500;
	stepTestFull[3197]:=49.500;
	stepTestFull[3198]:=49.500;
	stepTestFull[3199]:=49.500;
	stepTestFull[3200]:=49.500;
	stepTestFull[3201]:=49.500;
	stepTestFull[3202]:=49.500;
	stepTestFull[3203]:=49.500;
	stepTestFull[3204]:=49.500;
	stepTestFull[3205]:=49.500;
	stepTestFull[3206]:=49.500;
	stepTestFull[3207]:=49.500;
	stepTestFull[3208]:=49.500;
	stepTestFull[3209]:=49.500;
	stepTestFull[3210]:=49.500;
	stepTestFull[3211]:=49.500;
	stepTestFull[3212]:=49.500;
	stepTestFull[3213]:=49.500;
	stepTestFull[3214]:=49.500;
	stepTestFull[3215]:=49.500;
	stepTestFull[3216]:=49.500;
	stepTestFull[3217]:=49.500;
	stepTestFull[3218]:=49.500;
	stepTestFull[3219]:=49.500;
	stepTestFull[3220]:=49.500;
	stepTestFull[3221]:=49.500;
	stepTestFull[3222]:=49.500;
	stepTestFull[3223]:=49.500;
	stepTestFull[3224]:=49.500;
	stepTestFull[3225]:=49.500;
	stepTestFull[3226]:=49.500;
	stepTestFull[3227]:=49.500;
	stepTestFull[3228]:=49.500;
	stepTestFull[3229]:=49.500;
	stepTestFull[3230]:=49.500;
	stepTestFull[3231]:=49.500;
	stepTestFull[3232]:=49.500;
	stepTestFull[3233]:=49.500;
	stepTestFull[3234]:=49.500;
	stepTestFull[3235]:=49.500;
	stepTestFull[3236]:=49.500;
	stepTestFull[3237]:=49.500;
	stepTestFull[3238]:=49.500;
	stepTestFull[3239]:=49.500;
	stepTestFull[3240]:=49.500;
	stepTestFull[3241]:=49.500;
	stepTestFull[3242]:=49.500;
	stepTestFull[3243]:=49.500;
	stepTestFull[3244]:=49.500;
	stepTestFull[3245]:=49.500;
	stepTestFull[3246]:=49.500;
	stepTestFull[3247]:=49.500;
	stepTestFull[3248]:=49.500;
	stepTestFull[3249]:=49.500;
	stepTestFull[3250]:=49.500;
	stepTestFull[3251]:=49.500;
	stepTestFull[3252]:=49.500;
	stepTestFull[3253]:=49.500;
	stepTestFull[3254]:=49.500;
	stepTestFull[3255]:=49.500;
	stepTestFull[3256]:=49.500;
	stepTestFull[3257]:=49.500;
	stepTestFull[3258]:=49.500;
	stepTestFull[3259]:=49.500;
	stepTestFull[3260]:=49.500;
	stepTestFull[3261]:=49.500;
	stepTestFull[3262]:=49.500;
	stepTestFull[3263]:=49.500;
	stepTestFull[3264]:=49.500;
	stepTestFull[3265]:=49.500;
	stepTestFull[3266]:=49.500;
	stepTestFull[3267]:=49.500;
	stepTestFull[3268]:=49.500;
	stepTestFull[3269]:=49.500;
	stepTestFull[3270]:=49.500;
	stepTestFull[3271]:=49.500;
	stepTestFull[3272]:=49.500;
	stepTestFull[3273]:=49.500;
	stepTestFull[3274]:=49.500;
	stepTestFull[3275]:=49.500;
	stepTestFull[3276]:=49.500;
	stepTestFull[3277]:=49.500;
	stepTestFull[3278]:=49.500;
	stepTestFull[3279]:=49.500;
	stepTestFull[3280]:=49.500;
	stepTestFull[3281]:=49.500;
	stepTestFull[3282]:=49.500;
	stepTestFull[3283]:=49.500;
	stepTestFull[3284]:=49.500;
	stepTestFull[3285]:=49.500;
	stepTestFull[3286]:=49.500;
	stepTestFull[3287]:=49.500;
	stepTestFull[3288]:=49.500;
	stepTestFull[3289]:=49.500;
	stepTestFull[3290]:=49.500;
	stepTestFull[3291]:=49.500;
	stepTestFull[3292]:=49.500;
	stepTestFull[3293]:=49.500;
	stepTestFull[3294]:=49.500;
	stepTestFull[3295]:=49.500;
	stepTestFull[3296]:=49.500;
	stepTestFull[3297]:=49.500;
	stepTestFull[3298]:=49.500;
	stepTestFull[3299]:=49.500;
	stepTestFull[3300]:=49.500;
	stepTestFull[3301]:=49.500;
	stepTestFull[3302]:=49.500;
	stepTestFull[3303]:=49.500;
	stepTestFull[3304]:=49.500;
	stepTestFull[3305]:=49.500;
	stepTestFull[3306]:=49.500;
	stepTestFull[3307]:=49.500;
	stepTestFull[3308]:=49.500;
	stepTestFull[3309]:=49.500;
	stepTestFull[3310]:=49.500;
	stepTestFull[3311]:=49.500;
	stepTestFull[3312]:=49.500;
	stepTestFull[3313]:=49.500;
	stepTestFull[3314]:=49.500;
	stepTestFull[3315]:=49.500;
	stepTestFull[3316]:=49.500;
	stepTestFull[3317]:=49.500;
	stepTestFull[3318]:=49.500;
	stepTestFull[3319]:=49.500;
	stepTestFull[3320]:=49.500;
	stepTestFull[3321]:=49.500;
	stepTestFull[3322]:=49.500;
	stepTestFull[3323]:=49.500;
	stepTestFull[3324]:=49.500;
	stepTestFull[3325]:=49.500;
	stepTestFull[3326]:=49.500;
	stepTestFull[3327]:=49.500;
	stepTestFull[3328]:=49.500;
	stepTestFull[3329]:=49.500;
	stepTestFull[3330]:=50.000;
	stepTestFull[3331]:=50.000;
	stepTestFull[3332]:=50.000;
	stepTestFull[3333]:=50.000;
	stepTestFull[3334]:=50.000;
	stepTestFull[3335]:=50.000;
	stepTestFull[3336]:=50.000;
	stepTestFull[3337]:=50.000;
	stepTestFull[3338]:=50.000;
	stepTestFull[3339]:=50.000;
	stepTestFull[3340]:=50.000;
	stepTestFull[3341]:=50.000;
	stepTestFull[3342]:=50.000;
	stepTestFull[3343]:=50.000;
	stepTestFull[3344]:=50.000;
	stepTestFull[3345]:=50.000;
	stepTestFull[3346]:=50.000;
	stepTestFull[3347]:=50.000;
	stepTestFull[3348]:=50.000;
	stepTestFull[3349]:=50.000;
	stepTestFull[3350]:=50.000;
	stepTestFull[3351]:=50.000;
	stepTestFull[3352]:=50.000;
	stepTestFull[3353]:=50.000;
	stepTestFull[3354]:=50.000;
	stepTestFull[3355]:=50.000;
	stepTestFull[3356]:=50.000;
	stepTestFull[3357]:=50.000;
	stepTestFull[3358]:=50.000;
	stepTestFull[3359]:=50.000;
```
